// ----------------------------------------------------------
// msg002 Message 02
// ----------------------------------------------------------
      SET   ;
      R     DB2697.DBX  140.7;
      =     DB2697.DBX  141.4;

      CLR   ;
      =     DB2697.DBX  142.7;

// ----------------------------------------------------------
// msg003 Message 03
// ----------------------------------------------------------
      SET   ;
      R     DB2697.DBX  200.7;
      =     DB2697.DBX  201.4;

      CLR   ;
      =     DB2697.DBX  202.7;

NETWORK
TITLE =Sequence organisation

      CLR   ;
      =     M    122.2;

// SFM supply ----------------------------------------------------------------

// analog value to SFM Heißwasser-Wärmetauscher1 TT01 -----------------------
      L     DB2693.DBD  146;
      T     DB1691.DBD 1122; // !!! insert correct SFM !!!

// sequencer ----------------------------------------------------------------
      A     DB1693.DBX   43.1;
      S     DB1693.DBX   97.3;

      CALL FC    40 (
           UnitNo                   := #UnitNo);

NETWORK
TITLE =Auto / Manual

      SET   ;
      AN    M    122.2;
      JC    MODE;
      AN    M    120.1;

// assign actuator mode
      AN    M    120.1;
      =     DB2690.DBX 1545.4;
      =     DB2690.DBX 1625.4;
      =     DB2690.DBX 1705.4;
      =     DB2690.DBX 1785.4;
      =     DB2690.DBX 1865.4;
      =     DB2690.DBX 1945.4;
      =     DB2690.DBX 2025.4;
      =     DB2690.DBX 2105.4;
      =     DB2690.DBX 2185.4;
      =     DB2690.DBX 2265.4;
      =     DB2690.DBX 2345.4;
      =     DB2690.DBX 2425.4;
      =     DB2690.DBX 2505.4;
      =     DB2690.DBX 2585.4;
      =     DB2690.DBX 2665.4;
      =     DB2690.DBX 2745.4;
      =     DB2690.DBX 2825.4;
      =     DB2690.DBX 2905.4;
      =     DB2690.DBX 2985.4;
      =     DB2690.DBX 3065.4;
      =     DB2690.DBX 3145.4;
      =     DB2690.DBX 3225.4;



MODE: SET   ;

NETWORK
TITLE =A9_RR1 Reinigungsrücklauf Anlage 9 zu Kreis 1
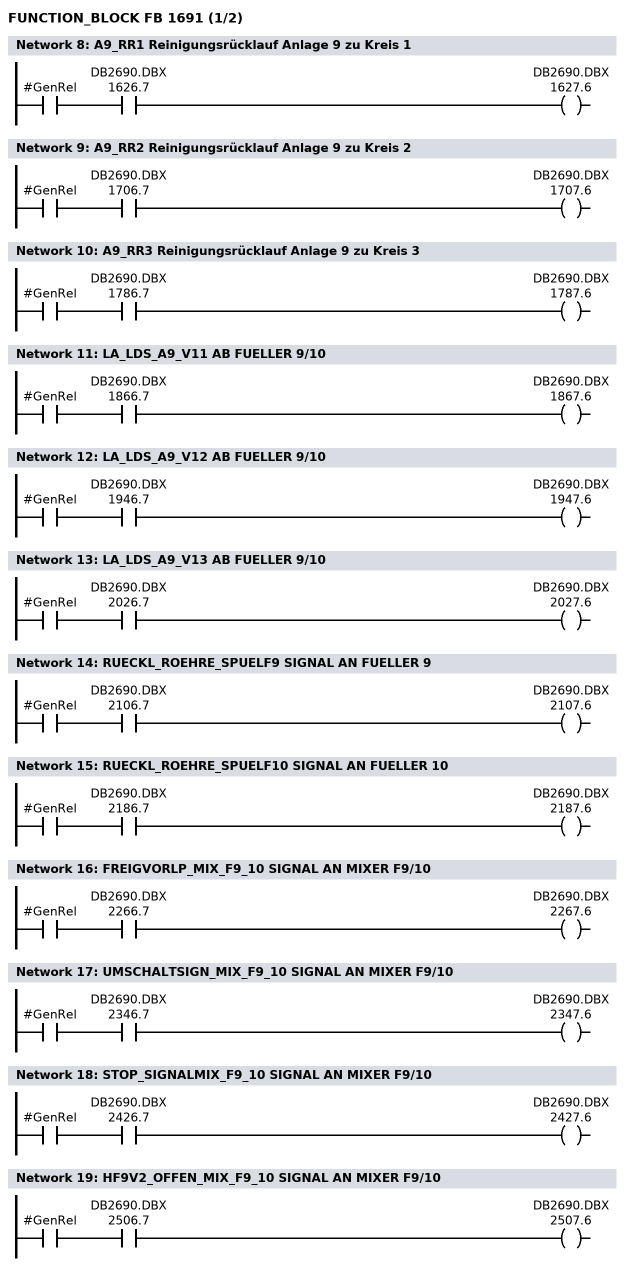

      A     #GenRel;
      A     DB2690.DBX 1626.7;
      =     DB2690.DBX 1627.6;
NETWORK
TITLE =A9_RR2 Reinigungsrücklauf Anlage 9 zu Kreis 2

      A     #GenRel;
      A     DB2690.DBX 1706.7;
      =     DB2690.DBX 1707.6;
NETWORK
TITLE =A9_RR3 Reinigungsrücklauf Anlage 9 zu Kreis 3

      A     #GenRel;
      A     DB2690.DBX 1786.7;
      =     DB2690.DBX 1787.6;
NETWORK
TITLE =LA_LDS_A9_V11 AB FUELLER 9/10

      A     #GenRel;
      A     DB2690.DBX 1866.7;
      =     DB2690.DBX 1867.6;
NETWORK
TITLE =LA_LDS_A9_V12 AB FUELLER 9/10

      A     #GenRel;
      A     DB2690.DBX 1946.7;
      =     DB2690.DBX 1947.6;
NETWORK
TITLE =LA_LDS_A9_V13 AB FUELLER 9/10

      A     #GenRel;
      A     DB2690.DBX 2026.7;
      =     DB2690.DBX 2027.6;
NETWORK
TITLE =RUECKL_ROEHRE_SPUELF9 SIGNAL AN FUELLER 9

      A     #GenRel;
      A     DB2690.DBX 2106.7;
      =     DB2690.DBX 2107.6;
NETWORK
TITLE =RUECKL_ROEHRE_SPUELF10 SIGNAL AN FUELLER 10

      A     #GenRel;
      A     DB2690.DBX 2186.7;
      =     DB2690.DBX 2187.6;
NETWORK
TITLE =FREIGVORLP_MIX_F9_10 SIGNAL AN MIXER F9/10

      A     #GenRel;
      A     DB2690.DBX 2266.7;
      =     DB2690.DBX 2267.6;
NETWORK
TITLE =UMSCHALTSIGN_MIX_F9_10 SIGNAL AN MIXER F9/10

      A     #GenRel;
      A     DB2690.DBX 2346.7;
      =     DB2690.DBX 2347.6;
NETWORK
TITLE =STOP_SIGNALMIX_F9_10 SIGNAL AN MIXER F9/10

      A     #GenRel;
      A     DB2690.DBX 2426.7;
      =     DB2690.DBX 2427.6;
NETWORK
TITLE =HF9V2_OFFEN_MIX_F9_10 SIGNAL AN MIXER F9/10

      A     #GenRel;
      A     DB2690.DBX 2506.7;
      =     DB2690.DBX 2507.6;
NETWORK
TITLE =FREIGVORLP_KASK_F9_10 SIGNAL AN MIXER F9/10
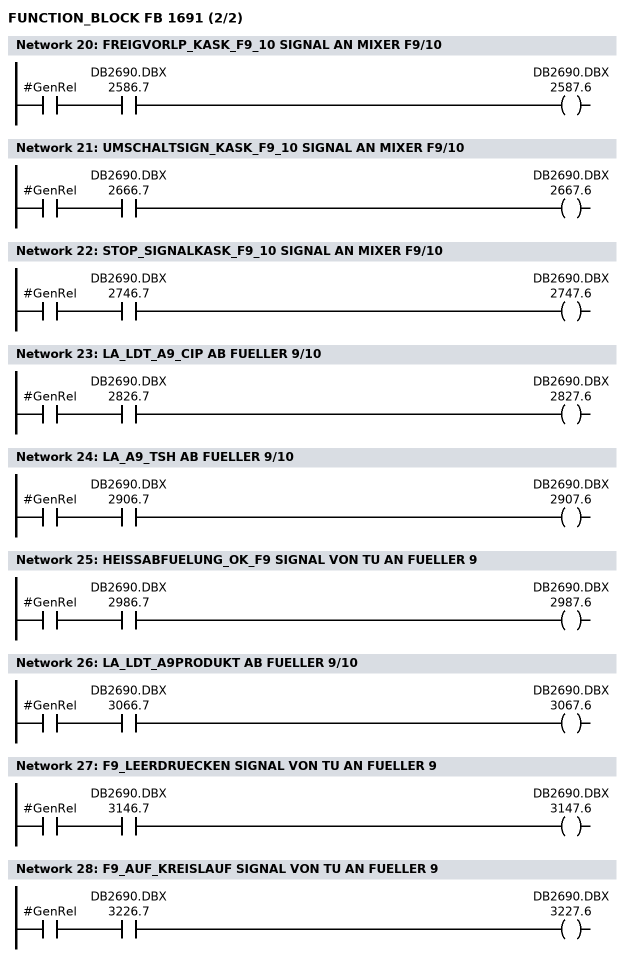

      A     #GenRel;
      A     DB2690.DBX 2586.7;
      =     DB2690.DBX 2587.6;
NETWORK
TITLE =UMSCHALTSIGN_KASK_F9_10 SIGNAL AN MIXER F9/10

      A     #GenRel;
      A     DB2690.DBX 2666.7;
      =     DB2690.DBX 2667.6;
NETWORK
TITLE =STOP_SIGNALKASK_F9_10 SIGNAL AN MIXER F9/10

      A     #GenRel;
      A     DB2690.DBX 2746.7;
      =     DB2690.DBX 2747.6;
NETWORK
TITLE =LA_LDT_A9_CIP AB FUELLER 9/10

      A     #GenRel;
      A     DB2690.DBX 2826.7;
      =     DB2690.DBX 2827.6;
NETWORK
TITLE =LA_A9_TSH AB FUELLER 9/10

      A     #GenRel;
      A     DB2690.DBX 2906.7;
      =     DB2690.DBX 2907.6;
NETWORK
TITLE =HEISSABFUELUNG_OK_F9 SIGNAL VON TU AN FUELLER 9

      A     #GenRel;
      A     DB2690.DBX 2986.7;
      =     DB2690.DBX 2987.6;
NETWORK
TITLE =LA_LDT_A9PRODUKT AB FUELLER 9/10

      A     #GenRel;
      A     DB2690.DBX 3066.7;
      =     DB2690.DBX 3067.6;
NETWORK
TITLE =F9_LEERDRUECKEN SIGNAL VON TU AN FUELLER 9

      A     #GenRel;
      A     DB2690.DBX 3146.7;
      =     DB2690.DBX 3147.6;
NETWORK
TITLE =F9_AUF_KREISLAUF SIGNAL VON TU AN FUELLER 9

      A     #GenRel;
      A     DB2690.DBX 3226.7;
      =     DB2690.DBX 3227.6;
END_FUNCTION_BLOCK

FUNCTION_BLOCK FB 1700
TITLE =U070: Abfüllanlage 10
FAMILY : BOTEC_F1
NAME : U070A
VERSION : 2.1


VAR_TEMP
  EStopOK : BOOL ;	//auxiliary flag
  CIP : BOOL ;	//CIP Program Selected
  xTmp : BOOL ;	//Temporary Bool(free for general use)
  DummyBool : BOOL ;	//Temporary Bool(free for general use)
  UnitNo : INT ;	//unit number
  UnitFB : INT ;	//unit expansion FB number
  rTmp : REAL ;	//Temporary REAL (free for general use)
  iTmp : INT ;	//Temporary INT (free for general use)
  DummyInt : INT ;	//Temporary INT (free for general use)
  dTmp : DINT ;	//Temporary DINT (free for general use)
END_VAR
BEGIN
NETWORK
TITLE =general

      CLR   ;
      =     #xTmp;
      =     #EStopOK;

      L     DB1700.DBW    0;
      T     #UnitNo;
      L     DB1700.DBW    2;
      T     #UnitFB;

NETWORK
TITLE =Universal value

      NOP   0;
// unv001 UnV 001 Process Status
      CALL FC    27 (
           UnitNo                   := #UnitNo,
           UnVRec                   := DB2705.unv001,
           ValExt                   := DB2705.DBD  234);

// unv002 UnV 002 Universal Value 02
      CALL FC    27 (
           UnitNo                   := #UnitNo,
           UnVRec                   := DB2705.unv002,
           ValExt                   := DB2705.DBD  362);

// unv003 UnV 003 Universal Value 03
      CALL FC    27 (
           UnitNo                   := #UnitNo,
           UnVRec                   := DB2705.unv003,
           ValExt                   := DB2705.DBD  490);

// unv004 UnV 004 Universal Value 04
      CALL FC    27 (
           UnitNo                   := #UnitNo,
           UnVRec                   := DB2705.unv004,
           ValExt                   := DB2705.DBD  618);

NETWORK
TITLE =special inputs

      NOP   0;
// LS_LLL_A10 SpI 001 LS_LLL_A10
      CALL FC    14 (
           UnitNo                   := #UnitNo,
           SpIRec                   := DB2701.LS_LLL_A10,
           SpIBit                   := I     62.3);

// TS_HL_ANL10 SpI 002 TS_HL_ANL10
      CALL FC    14 (
           UnitNo                   := #UnitNo,
           SpIRec                   := DB2701.TS_HL_ANL10,
           SpIBit                   := I     62.1);

// DT_A10_START SpI 003 DT_A10_START
      CALL FC    14 (
           UnitNo                   := #UnitNo,
           SpIRec                   := DB2701.DT_A10_START,
           SpIBit                   := I     53.4);

// DT_A10_STOP SpI 004 DT_A10_STOP
      CALL FC    14 (
           UnitNo                   := #UnitNo,
           SpIRec                   := DB2701.DT_A10_STOP,
           SpIBit                   := I     53.5);

// BETRIEB_F10 SpI 005 BETRIEB_F10
      CALL FC    14 (
           UnitNo                   := #UnitNo,
           SpIRec                   := DB2701.BETRIEB_F10,
           SpIBit                   := I     62.5);

// BETRIEB_MIX_LKASKADE_F10 SpI 006 BETRIEB_MIX_LKASKADE_F10
      CALL FC    14 (
           UnitNo                   := #UnitNo,
           SpIRec                   := DB2701.BETRIEB_MIX_LKASKADE_F10,
           SpIBit                   := I     62.7);

// KASK_ANFORDERUNG_PUMPE SpI 007 KASK_ANFORDERUNG_PUMPE
      CALL FC    14 (
           UnitNo                   := #UnitNo,
           SpIRec                   := DB2701.KASK_ANFORDERUNG_PUMPE,
           SpIBit                   := I    123.3);

// RM_RWPA10 SpI 008 RM_RWPA10
      CALL FC    14 (
           UnitNo                   := #UnitNo,
           SpIRec                   := DB2701.RM_RWPA10,
           SpIBit                   := I    123.4);

// KAS_WEGFREIGABE_10_L9 SpI 009 KAS_WEGFREIGABE_10_L9
      CALL FC    14 (
           UnitNo                   := #UnitNo,
           SpIRec                   := DB2701.KAS_WEGFREIGABE_10_L9,
           SpIBit                   := I    123.5);

// KAS_WEGFREIGABE_10_L10 SpI 010 KAS_WEGFREIGABE_10_L10
      CALL FC    14 (
           UnitNo                   := #UnitNo,
           SpIRec                   := DB2701.KAS_WEGFREIGABE_10_L10,
           SpIBit                   := I    123.6);

NETWORK
TITLE =messages

      NOP   0;
// msg001 Msg 001 Message 01
      CALL FC    16 (
           UnitNo                   := #UnitNo,
           MsgRec                   := DB2707.msg001,
           MsgBit                   := DB2707.DBX   82.7);

// msg002 Msg 002 Message 02
      CALL FC    16 (
           UnitNo                   := #UnitNo,
           MsgRec                   := DB2707.msg002,
           MsgBit                   := DB2707.DBX  142.7);

// msg003 Msg 003 Message 03
      CALL FC    16 (
           UnitNo                   := #UnitNo,
           MsgRec                   := DB2707.msg003,
           MsgBit                   := DB2707.DBX  202.7);

NETWORK
TITLE =unit supply

      UC    FB [#UnitFB];

NETWORK
TITLE =A10_RR1  Reinigungsrücklauf Anlage 10 zu Kreis 1
// Act 020
// Box           : VSRR1-3
// Input address : I84.6
// Output address: Q84.6
      CALL FC    70 (
           UnitNo                   := #UnitNo,
           ActRec                   := DB2700.A10_RR1,
           Typ                      := 1,
           FBa                      := #xTmp,
           FBa2                     := I     84.6,
           Out                      := Q     84.6);

NETWORK
TITLE =A10_RR2  Reinigungsrücklauf Anlage 10 zu Kreis 2
// Act 021
// Box           : VSRR1-3
// Input address : I84.7
// Output address: Q84.7
      CALL FC    70 (
           UnitNo                   := #UnitNo,
           ActRec                   := DB2700.A10_RR2,
           Typ                      := 1,
           FBa                      := #xTmp,
           FBa2                     := I     84.7,
           Out                      := Q     84.7);

NETWORK
TITLE =A10_RR3  Reinigungsrücklauf Anlage 10 zu Kreis 3
// Act 022
// Box           : VSRR1-3
// Input address : I85.0
// Output address: Q85.0
      CALL FC    70 (
           UnitNo                   := #UnitNo,
           ActRec                   := DB2700.A10_RR3,
           Typ                      := 1,
           FBa                      := #xTmp,
           FBa2                     := I     85.0,
           Out                      := Q     85.0);

NETWORK
TITLE =LA_LDS_A10V13  LA_LDS_A10V13
// Act 023
// Box           : S8 U8.2
// Input address : I53.1
// Output address: Q110.0
      CALL FC    70 (
           UnitNo                   := #UnitNo,
           ActRec                   := DB2700.LA_LDS_A10V13,
           Typ                      := 0,
           FBa                      := #xTmp,
           FBa2                     := I     53.1,
           Out                      := Q    110.0);

NETWORK
TITLE =LA_LDT_A10PRODUKT  LA_LDT_A10PRODUKT
// Act 024
// Box           : S8 U8.2
// Input address : I53.2
// Output address: Q110.1
      CALL FC    70 (
           UnitNo                   := #UnitNo,
           ActRec                   := DB2700.LA_LDT_A10PRODUKT,
           Typ                      := 0,
           FBa                      := #xTmp,
           FBa2                     := I     53.2,
           Out                      := Q    110.1);

NETWORK
TITLE =LA_LDT_A10CIP  LA_LDT_A10CIP
// Act 025
// Box           : S8 U8.2
// Input address : I53.3
// Output address: Q110.2
      CALL FC    70 (
           UnitNo                   := #UnitNo,
           ActRec                   := DB2700.LA_LDT_A10CIP,
           Typ                      := 0,
           FBa                      := #xTmp,
           FBa2                     := I     53.3,
           Out                      := Q    110.2);

NETWORK
TITLE =LA_A10TSH  LA_A10TSH
// Act 026
// Box           : S8 U8.2
// Output address: Q110.3
      CALL FC    70 (
           UnitNo                   := #UnitNo,
           ActRec                   := DB2700.LA_A10TSH,
           Typ                      := 0,
           FBa                      := #xTmp,
           FBa2                     := #xTmp,
           Out                      := Q    110.3);

NETWORK
TITLE =LA_STOERUNG_CIP  LA_STOERUNG_CIP
// Act 027
// Box           : S8 U8.2
// Output address: Q110.4
      CALL FC    70 (
           UnitNo                   := #UnitNo,
           ActRec                   := DB2700.LA_STOERUNG_CIP,
           Typ                      := 0,
           FBa                      := #xTmp,
           FBa2                     := #xTmp,
           Out                      := Q    110.4);

NETWORK
TITLE =LA_ALARML9_10  LA_ALARML9_10
// Act 028
// Box           : S8 U8.2
// Output address: Q110.5
      CALL FC    70 (
           UnitNo                   := #UnitNo,
           ActRec                   := DB2700.LA_ALARML9_10,
           Typ                      := 0,
           FBa                      := #xTmp,
           FBa2                     := #xTmp,
           Out                      := Q    110.5);

NETWORK
TITLE =LA_LDS_A10V11  LA_LDS_A10V11
// Act 029
// Box           : S8 U8.2
// Input address : I52.7
// Output address: Q110.6
      CALL FC    70 (
           UnitNo                   := #UnitNo,
           ActRec                   := DB2700.LA_LDS_A10V11,
           Typ                      := 0,
           FBa                      := #xTmp,
           FBa2                     := I     52.7,
           Out                      := Q    110.6);

NETWORK
TITLE =LA_LDS_A10V12  LA_LDS_A10V12
// Act 030
// Box           : S8 U8.2
// Input address : I53.0
// Output address: Q110.7
      CALL FC    70 (
           UnitNo                   := #UnitNo,
           ActRec                   := DB2700.LA_LDS_A10V12,
           Typ                      := 0,
           FBa                      := #xTmp,
           FBa2                     := I     53.0,
           Out                      := Q    110.7);

NETWORK
TITLE =UMSCHALTSIGN_KASK_F9_10  UMSCHALTSIGN_KASK_F9_10
// Act 031
// Box           : S8 U8.2
// Output address: Q41.6
      CALL FC    70 (
           UnitNo                   := #UnitNo,
           ActRec                   := DB2700.UMSCHALTSIGN_KASK_F9_10,
           Typ                      := 0,
           FBa                      := #xTmp,
           FBa2                     := #xTmp,
           Out                      := Q     41.6);

NETWORK
TITLE =STOP_SIGNALKASK_F9_10  STOP_SIGNALKASK_F9_10
// Act 032
// Box           : S8 U8.2
// Output address: Q41.7
      CALL FC    70 (
           UnitNo                   := #UnitNo,
           ActRec                   := DB2700.STOP_SIGNALKASK_F9_10,
           Typ                      := 0,
           FBa                      := #xTmp,
           FBa2                     := #xTmp,
           Out                      := Q     41.7);

END_FUNCTION_BLOCK

FUNCTION_BLOCK FB 1701
TITLE =U070: Packaging Plant 10
FAMILY : BOTEC_F1
NAME : UniE
VERSION : 1.2


VAR_TEMP
  CIP : BOOL ;	//CIP active
  UNIM : BOOL ;	//Unit Not In Maintenance
  GenRel : BOOL ;	//general OK (emergency and maintenance OK)
  EStopOK : BOOL ;	//emergency OK
  UnitNo : INT ;	//unit number
  xTmp : BOOL ;	//Temporary Bool
  iTmp : INT ;	//Temporary INT
  rTmp : REAL ;	//Temporary REAL
  dTmp : DINT ;	//Temporary DINT (free for general use)
  RetValInt : INT ;	//return value
END_VAR
BEGIN
NETWORK
TITLE =General

      SET   ;
// Simulation ---------------------------------------------------------------
      A     DB1701.DBX 1357.7;
      CC    FB  1709; // "U070Sim"
      A     DB1701.DBX   17.3;
      =     DB1701.DBX 1357.7; //Help bit for simulation

// get unit number ----------------------------------------------------------
      L     DB1700.DBW    0;
      T     #UnitNo;

// CIP ----------------------------------------------------------------------
      L     DB1701.DBD   54;
      L     0;
      <D    ;
      =     #CIP;

// emergency OK -------------------------------------------------------------
      A     DB1705.DBX   27.0; //Emergency Stop OK
      =     #EStopOK;

// Write Unit in Maintenance ------------------------------------------------

      AN    DB1701.DBX   69.7;
      =     #UNIM;

// emergency and maintenance OK ---------------------------------------------
      A     #EStopOK;
      A     #UNIM;
      =     #GenRel;

// communication ------------------------------------------------------------
      UC    FB  1705; // U070Com

NETWORK
TITLE =Universal Value

      NOP   0;

// ----------------------------------------------------------
// unv001 Process Status
// ----------------------------------------------------------
// process value to UnV
//      L     0.000000e+000
//      T     "U070UnVD".unv001.ValExt

// ----------------------------------------------------------
// unv002 Universal Value 02
// ----------------------------------------------------------
// process value to UnV
//      L     0.000000e+000
//      T     "U070UnVD".unv002.ValExt

// ----------------------------------------------------------
// unv003 Universal Value 03
// ----------------------------------------------------------
// process value to UnV
//      L     0.000000e+000
//      T     "U070UnVD".unv003.ValExt

// ----------------------------------------------------------
// unv004 Universal Value 04
// ----------------------------------------------------------
// process value to UnV
//      L     0.000000e+000
//      T     "U070UnVD".unv004.ValExt

NETWORK
TITLE =Special Input

      NOP   0;

// ----------------------------------------------------------
// LS_LLL_A10 SIGNAL VON FUELLER 10
// ----------------------------------------------------------
//      A     "U070SeqD".Seq.Step0
//      =     "U070SpID".LS_LLL_A10.EAl
//      SET
//      =     "U070SpID".LS_LLL_A10.Pre

// ----------------------------------------------------------
// TS_HL_ANL10
// ----------------------------------------------------------
//      A     "U070SeqD".Seq.Step0
//      =     "U070SpID".TS_HL_ANL10.EAl
//      SET
//      =     "U070SpID".TS_HL_ANL10.Pre

// ----------------------------------------------------------
// DT_A10_START AB FUELLER 9/10
// ----------------------------------------------------------
//      CLR
//      =     "U070SpID".DT_A10_START.EAl
//      =     "U070SpID".DT_A10_START.Pre

// ----------------------------------------------------------
// DT_A10_STOP AB FUELLER 9/10
// ----------------------------------------------------------
//      CLR
//      =     "U070SpID".DT_A10_STOP.EAl
//      =     "U070SpID".DT_A10_STOP.Pre

// ----------------------------------------------------------
// BETRIEB_F10 SIGNAL VON FUELLER 10
// ----------------------------------------------------------
//      CLR
//      =     "U070SpID".BETRIEB_F10.EAl
//      =     "U070SpID".BETRIEB_F10.Pre

// ----------------------------------------------------------
// BETRIEB_MIX_LKASKADE_F10 SIGNAL VON FUELLER 10
// ----------------------------------------------------------
//      CLR
//      =     "U070SpID".BETRIEB_MIX_LKASKADE_F10.EAl
//      =     "U070SpID".BETRIEB_MIX_LKASKADE_F10.Pre

// ----------------------------------------------------------
// KASK_ANFORDERUNG_PUMPE SIGNAL VON KASKADE
// ----------------------------------------------------------
//      CLR
//      =     "U070SpID".KASK_ANFORDERUNG_PUMPE.EAl
//      =     "U070SpID".KASK_ANFORDERUNG_PUMPE.Pre

// ----------------------------------------------------------
// RM_RWPA10 SIGNAL VON MIXER F9/10
// ----------------------------------------------------------
      A     DB1701.DBX 1230.3;
      A     DB1701.DBX 1262.3;
      =     DB2701.DBX  501.4;
      =     DB2701.DBX  501.5;

// ----------------------------------------------------------
// KAS_WEGFREIGABE_10_L9 SIGNAL VON KASKADE F9/10
// ----------------------------------------------------------
//      CLR
//      =     "U070SpID".KAS_WEGFREIGABE_10_L9.EAl
//      =     "U070SpID".KAS_WEGFREIGABE_10_L9.Pre

// ----------------------------------------------------------
// KAS_WEGFREIGABE_10_L10 SIGNAL VON KASKADE F9/10
// ----------------------------------------------------------
//      CLR
//      =     "U070SpID".KAS_WEGFREIGABE_10_L10.EAl
//      =     "U070SpID".KAS_WEGFREIGABE_10_L10.Pre

NETWORK
TITLE =Messages

      NOP   0;

// ----------------------------------------------------------
// msg001 Message 01
// ----------------------------------------------------------
      SET   ;
      R     DB2707.DBX   80.7;
      =     DB2707.DBX   81.4;

      CLR   ;
      =     DB2707.DBX   82.7;

// ----------------------------------------------------------
// msg002 Message 02
// ----------------------------------------------------------
      SET   ;
      R     DB2707.DBX  140.7;
      =     DB2707.DBX  141.4;

      CLR   ;
      =     DB2707.DBX  142.7;

// ----------------------------------------------------------
// msg003 Message 03
// ----------------------------------------------------------
      SET   ;
      R     DB2707.DBX  200.7;
      =     DB2707.DBX  201.4;

      CLR   ;
      =     DB2707.DBX  202.7;

NETWORK
TITLE =Sequence organisation

      CLR   ;
      =     M    122.2;

// SFM supply ----------------------------------------------------------------

// sequencer ----------------------------------------------------------------
      A     DB1703.DBX   43.1;
      S     DB1703.DBX   97.3;

      CALL FC    40 (
           UnitNo                   := #UnitNo);

NETWORK
TITLE =Auto / Manual

      SET   ;
      AN    M    122.2;
      JC    MODE;
      AN    M    120.1;

// assign actuator mode
      AN    M    120.1;
      =     DB2700.DBX 1625.4;
      =     DB2700.DBX 1705.4;
      =     DB2700.DBX 1785.4;
      =     DB2700.DBX 1865.4;
      =     DB2700.DBX 1945.4;
      =     DB2700.DBX 2025.4;
      =     DB2700.DBX 2105.4;
      =     DB2700.DBX 2185.4;
      =     DB2700.DBX 2265.4;
      =     DB2700.DBX 2345.4;
      =     DB2700.DBX 2425.4;
      =     DB2700.DBX 2505.4;
      =     DB2700.DBX 2585.4;

MODE: SET   ;

NETWORK
TITLE =A10_RR1 Reinigungsrücklauf Anlage 10 zu Kreis 1
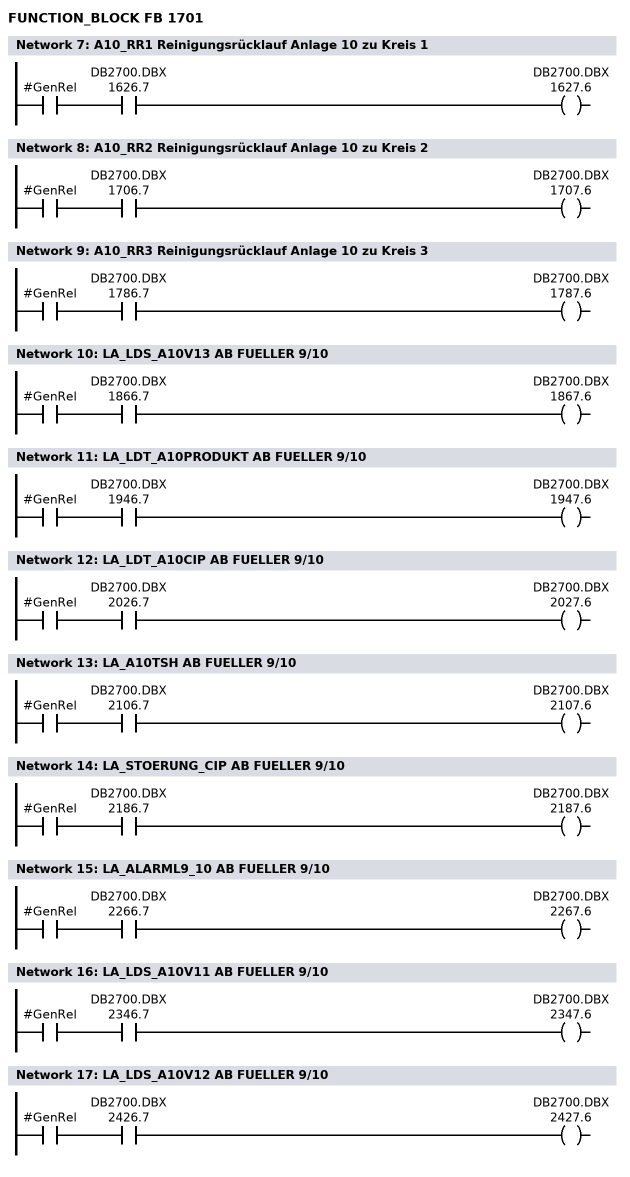

      A     #GenRel;
      A     DB2700.DBX 1626.7;
      =     DB2700.DBX 1627.6;
NETWORK
TITLE =A10_RR2 Reinigungsrücklauf Anlage 10 zu Kreis 2

      A     #GenRel;
      A     DB2700.DBX 1706.7;
      =     DB2700.DBX 1707.6;
NETWORK
TITLE =A10_RR3 Reinigungsrücklauf Anlage 10 zu Kreis 3

      A     #GenRel;
      A     DB2700.DBX 1786.7;
      =     DB2700.DBX 1787.6;
NETWORK
TITLE =LA_LDS_A10V13 AB FUELLER 9/10

      A     #GenRel;
      A     DB2700.DBX 1866.7;
      =     DB2700.DBX 1867.6;
NETWORK
TITLE =LA_LDT_A10PRODUKT AB FUELLER 9/10

      A     #GenRel;
      A     DB2700.DBX 1946.7;
      =     DB2700.DBX 1947.6;
NETWORK
TITLE =LA_LDT_A10CIP AB FUELLER 9/10

      A     #GenRel;
      A     DB2700.DBX 2026.7;
      =     DB2700.DBX 2027.6;
NETWORK
TITLE =LA_A10TSH AB FUELLER 9/10

      A     #GenRel;
      A     DB2700.DBX 2106.7;
      =     DB2700.DBX 2107.6;
NETWORK
TITLE =LA_STOERUNG_CIP AB FUELLER 9/10

      A     #GenRel;
      A     DB2700.DBX 2186.7;
      =     DB2700.DBX 2187.6;
NETWORK
TITLE =LA_ALARML9_10 AB FUELLER 9/10

      A     #GenRel;
      A     DB2700.DBX 2266.7;
      =     DB2700.DBX 2267.6;
NETWORK
TITLE =LA_LDS_A10V11 AB FUELLER 9/10

      A     #GenRel;
      A     DB2700.DBX 2346.7;
      =     DB2700.DBX 2347.6;
NETWORK
TITLE =LA_LDS_A10V12 AB FUELLER 9/10

      A     #GenRel;
      A     DB2700.DBX 2426.7;
      =     DB2700.DBX 2427.6;
END_FUNCTION_BLOCK

FUNCTION_BLOCK FB 1710
TITLE =U071: Abfüllanlage 11
FAMILY : BOTEC_F1
NAME : U071A
VERSION : 2.1


VAR_TEMP
  EStopOK : BOOL ;	//auxiliary flag
  CIP : BOOL ;	//CIP Program Selected
  xTmp : BOOL ;	//Temporary Bool(free for general use)
  DummyBool : BOOL ;	//Temporary Bool(free for general use)
  UnitNo : INT ;	//unit number
  UnitFB : INT ;	//unit expansion FB number
  rTmp : REAL ;	//Temporary REAL (free for general use)
  iTmp : INT ;	//Temporary INT (free for general use)
  DummyInt : INT ;	//Temporary INT (free for general use)
  dTmp : DINT ;	//Temporary DINT (free for general use)
END_VAR
BEGIN
NETWORK
TITLE =general

      CLR   ;
      =     #xTmp;
      =     #EStopOK;

      L     DB1710.DBW    0;
      T     #UnitNo;
      L     DB1710.DBW    2;
      T     #UnitFB;

NETWORK
TITLE =Universal value

      NOP   0;
// unv001 UnV 001 Process Status
      CALL FC    27 (
           UnitNo                   := #UnitNo,
           UnVRec                   := DB2715.unv001,
           ValExt                   := DB2715.DBD  234);

// unv002 UnV 002 Universal Value 02
      CALL FC    27 (
           UnitNo                   := #UnitNo,
           UnVRec                   := DB2715.unv002,
           ValExt                   := DB2715.DBD  362);

// unv003 UnV 003 Universal Value 03
      CALL FC    27 (
           UnitNo                   := #UnitNo,
           UnVRec                   := DB2715.unv003,
           ValExt                   := DB2715.DBD  490);

// unv004 UnV 004 Universal Value 04
      CALL FC    27 (
           UnitNo                   := #UnitNo,
           UnVRec                   := DB2715.unv004,
           ValExt                   := DB2715.DBD  618);

NETWORK
TITLE =special inputs

      NOP   0;
// A9_FS1 SpI 001 geändert 07.11.01 A11 FS1 Stömungswächter
      CALL FC    14 (
           UnitNo                   := #UnitNo,
           SpIRec                   := DB2711.A9_FS1,
           SpIBit                   := I    177.0);

// A11_Fueller_laeuft SpI 002 Füller 11 läuft (Dauersignal)
      CALL FC    14 (
           UnitNo                   := #UnitNo,
           SpIRec                   := DB2711.A11_Fueller_laeuft,
           SpIBit                   := I    168.1);

// A11_Mixer_CIP_Bereit SpI 003 Mixer A 11 CIP-Bereitschaft (Dauersign)
      CALL FC    14 (
           UnitNo                   := #UnitNo,
           SpIRec                   := DB2711.A11_Mixer_CIP_Bereit,
           SpIBit                   := I    170.0);

// A11_Mixer_voll SpI 004 Mixer A 11 voll
      CALL FC    14 (
           UnitNo                   := #UnitNo,
           SpIRec                   := DB2711.A11_Mixer_voll,
           SpIBit                   := I    170.2);

// A11_Mixer_leer SpI 005 Mixer A 11 leer
      CALL FC    14 (
           UnitNo                   := #UnitNo,
           SpIRec                   := DB2711.A11_Mixer_leer,
           SpIBit                   := I    170.1);

// A11_Mixer_Anf_Sirup SpI 006 Mixer A 11 Anforderung Sirup
      CALL FC    14 (
           UnitNo                   := #UnitNo,
           SpIRec                   := DB2711.A11_Mixer_Anf_Sirup,
           SpIBit                   := I    170.3);

// A11_Fueller_CIP_Bereit SpI 007 Füller 11 CIP-Bereitschaft (Dauer)
      CALL FC    14 (
           UnitNo                   := #UnitNo,
           SpIRec                   := DB2711.A11_Fueller_CIP_Bereit,
           SpIBit                   := I    168.0);

// A11_Fueller_leer SpI 011 Füller 11 leer (Impuls)
      CALL FC    14 (
           UnitNo                   := #UnitNo,
           SpIRec                   := DB2711.A11_Fueller_leer,
           SpIBit                   := I    168.2);

// All_Fueller_voll SpI 012 Füller 11 voll (Impuls)
      CALL FC    14 (
           UnitNo                   := #UnitNo,
           SpIRec                   := DB2711.All_Fueller_voll,
           SpIBit                   := I    168.3);

NETWORK
TITLE =messages

      NOP   0;
// msg001 Msg 001 Message 01
      CALL FC    16 (
           UnitNo                   := #UnitNo,
           MsgRec                   := DB2717.msg001,
           MsgBit                   := DB2717.DBX   82.7);

// msg002 Msg 002 Message 02
      CALL FC    16 (
           UnitNo                   := #UnitNo,
           MsgRec                   := DB2717.msg002,
           MsgBit                   := DB2717.DBX  142.7);

// msg003 Msg 003 Message 03
      CALL FC    16 (
           UnitNo                   := #UnitNo,
           MsgRec                   := DB2717.msg003,
           MsgBit                   := DB2717.DBX  202.7);

NETWORK
TITLE =unit supply

      UC    FB [#UnitFB];

NETWORK
TITLE =A11_RP1  A11RP1 Anlage 11 Reinigungsrücklaufpumpe
// Act 001
// Box           : S6 U6.3
// Input address : I6.3
// Output address: Q6.3
      CALL FC    70 (
           UnitNo                   := #UnitNo,
           ActRec                   := DB2710.A11_RP1,
           Typ                      := 1,
           FBa                      := #xTmp,
           FBa2                     := I      6.3,
           Out                      := Q      6.3);

NETWORK
TITLE =F11_Maschine_Start  Füller 11 Maschine_Start
// Act 002
// Box           : FM-A11
// Output address: Q168.0
      CALL FC    70 (
           UnitNo                   := #UnitNo,
           ActRec                   := DB2710.F11_Maschine_Start,
           Typ                      := 0,
           FBa                      := #xTmp,
           FBa2                     := #xTmp,
           Out                      := Q    168.0);

NETWORK
TITLE =F11_Maschine_Stop  Füller 11 Maschine_Stop
// Act 003
// Box           : FM-A11
// Output address: Q168.1
      CALL FC    70 (
           UnitNo                   := #UnitNo,
           ActRec                   := DB2710.F11_Maschine_Stop,
           Typ                      := 0,
           FBa                      := #xTmp,
           FBa2                     := #xTmp,
           Out                      := #xTmp);

NETWORK
TITLE =F11_CIP_Kreislauf_o_puls  Füller 11 CIP-Kreisl. ohne puls
// Act 010
// Box           : FM-A11
// Output address: Q168.2
      CALL FC    70 (
           UnitNo                   := #UnitNo,
           ActRec                   := DB2710.F11_CIP_Kreislauf_o_puls,
           Typ                      := 0,
           FBa                      := #xTmp,
           FBa2                     := #xTmp,
           Out                      := Q    168.2);

NETWORK
TITLE =F11_CIP_Kreislauf_m_puls  Füller 11 CIP-Kreisl. mit puls
// Act 011
// Box           : FM-A11
// Output address: Q168.3
      CALL FC    70 (
           UnitNo                   := #UnitNo,
           ActRec                   := DB2710.F11_CIP_Kreislauf_m_puls,
           Typ                      := 0,
           FBa                      := #xTmp,
           FBa2                     := #xTmp,
           Out                      := Q    168.3);

NETWORK
TITLE =F11_Randvollstellung  Füller 11 Randvollstellung Desinfektion
// Act 012
// Box           : FM-A11
// Output address: Q168.4
      CALL FC    70 (
           UnitNo                   := #UnitNo,
           ActRec                   := DB2710.F11_Randvollstellung,
           Typ                      := 0,
           FBa                      := #xTmp,
           FBa2                     := #xTmp,
           Out                      := Q    168.4);

NETWORK
TITLE =F11_Klarspuel_o_CIP_Beh  Füller 11 Klarspülen ohne CIP-Behälter
// Act 013
// Box           : FM-A11
// Output address: Q168.5
      CALL FC    70 (
           UnitNo                   := #UnitNo,
           ActRec                   := DB2710.F11_Klarspuel_o_CIP_Beh,
           Typ                      := 0,
           FBa                      := #xTmp,
           FBa2                     := #xTmp,
           Out                      := Q    168.5);

NETWORK
TITLE =F11_Ausschub_m_Steriluft  Füller 11 Ausschub mit Sterrielluft
// Act 014
// Box           : FM-A11
// Output address: Q168.6
      CALL FC    70 (
           UnitNo                   := #UnitNo,
           ActRec                   := DB2710.F11_Ausschub_m_Steriluft,
           Typ                      := 0,
           FBa                      := #xTmp,
           FBa2                     := #xTmp,
           Out                      := Q    168.6);

NETWORK
TITLE =F11_Ausschub_m_CO2  Füller 11 Ausschub mit CO2
// Act 015
// Box           : FM-A11
// Output address: Q168.7
      CALL FC    70 (
           UnitNo                   := #UnitNo,
           ActRec                   := DB2710.F11_Ausschub_m_CO2,
           Typ                      := 0,
           FBa                      := #xTmp,
           FBa2                     := #xTmp,
           Out                      := Q    168.7);

NETWORK
TITLE =F11_Grundstellung_IMP  F11_Grungstellung_IMPULS
// Act 016
// Box           : FM-A11
// Output address: Q169.0
      CALL FC    70 (
           UnitNo                   := #UnitNo,
           ActRec                   := DB2710.F11_Grundstellung_IMP,
           Typ                      := 0,
           FBa                      := #xTmp,
           FBa2                     := #xTmp,
           Out                      := Q    169.0);

NETWORK
TITLE =F11_Drainagestellung_IMP  F11_Drainagestellung_IMPULS
// Act 017
// Box           : FM-A11
// Output address: Q169.1
      CALL FC    70 (
           UnitNo                   := #UnitNo,
           ActRec                   := DB2710.F11_Drainagestellung_IMP,
           Typ                      := 0,
           FBa                      := #xTmp,
           FBa2                     := #xTmp,
           Out                      := Q    169.1);

NETWORK
TITLE =F11_Bypass_IMP  F11_BYPASS_IMPULS
// Act 018
// Box           : FM-A11
// Output address: Q169.2
      CALL FC    70 (
           UnitNo                   := #UnitNo,
           ActRec                   := DB2710.F11_Bypass_IMP,
           Typ                      := 0,
           FBa                      := #xTmp,
           FBa2                     := #xTmp,
           Out                      := Q    169.2);

NETWORK
TITLE =A11_RR1  A11RR1 Ventil CIP Rücklauf Kreis 1 Anlage 11
// Act 020
// Box           : VSRR6-11
// Input address : I28.3
// Output address: Q28.3
      CALL FC    70 (
           UnitNo                   := #UnitNo,
           ActRec                   := DB2710.A11_RR1,
           Typ                      := 1,
           FBa                      := #xTmp,
           FBa2                     := I     28.3,
           Out                      := Q     28.3);

NETWORK
TITLE =A11_RR2  A11RR2 Ventil CIP Rücklauf Kreis 2 Anlage 11
// Act 021
// Box           : VSRR6-11
// Input address : I28.4
// Output address: Q28.4
      CALL FC    70 (
           UnitNo                   := #UnitNo,
           ActRec                   := DB2710.A11_RR2,
           Typ                      := 1,
           FBa                      := #xTmp,
           FBa2                     := I     28.4,
           Out                      := Q     28.4);

NETWORK
TITLE =A11_RR3  A11RR3 Ventil CIP Rücklauf Kreis 3 Anlage 11
// Act 022
// Box           : VSRR6-11
// Input address : I28.5
// Output address: Q28.5
      CALL FC    70 (
           UnitNo                   := #UnitNo,
           ActRec                   := DB2710.A11_RR3,
           Typ                      := 1,
           FBa                      := #xTmp,
           FBa2                     := I     28.5,
           Out                      := Q     28.5);

NETWORK
TITLE =M11_Grundstellung_IMP  Mixer A11 Sign. als Impuls
// Act 023
// Box           : FM-A11
// Output address: Q170.0
      CALL FC    70 (
           UnitNo                   := #UnitNo,
           ActRec                   := DB2710.M11_Grundstellung_IMP,
           Typ                      := 0,
           FBa                      := #xTmp,
           FBa2                     := #xTmp,
           Out                      := Q    170.0);

NETWORK
TITLE =M11_Drainagestellung_IMP  Mixer A11 Sign. als Impuls
// Act 024
// Box           : FM-A11
// Output address: Q170.1
      CALL FC    70 (
           UnitNo                   := #UnitNo,
           ActRec                   := DB2710.M11_Drainagestellung_IMP,
           Typ                      := 0,
           FBa                      := #xTmp,
           FBa2                     := #xTmp,
           Out                      := Q    170.1);

NETWORK
TITLE =M11_Ausspritzen_o_Ablauf  Mixer A11 Sign. als Impuls
// Act 025
// Box           : FM-A11
// Output address: Q170.2
      CALL FC    70 (
           UnitNo                   := #UnitNo,
           ActRec                   := DB2710.M11_Ausspritzen_o_Ablauf,
           Typ                      := 0,
           FBa                      := #xTmp,
           FBa2                     := #xTmp,
           Out                      := Q    170.2);

NETWORK
TITLE =M11_Ausspritzen_m_Ablauf  Mixer A11 Sign. als Impuls
// Act 026
// Box           : FM-A11
// Output address: Q170.3
      CALL FC    70 (
           UnitNo                   := #UnitNo,
           ActRec                   := DB2710.M11_Ausspritzen_m_Ablauf,
           Typ                      := 0,
           FBa                      := #xTmp,
           FBa2                     := #xTmp,
           Out                      := Q    170.3);

NETWORK
TITLE =M11_Fluten_o_Ablauf  Mixer A11 Sign. als Impuls
// Act 027
// Box           : FM-A11
// Output address: Q170.4
      CALL FC    70 (
           UnitNo                   := #UnitNo,
           ActRec                   := DB2710.M11_Fluten_o_Ablauf,
           Typ                      := 0,
           FBa                      := #xTmp,
           FBa2                     := #xTmp,
           Out                      := Q    170.4);

NETWORK
TITLE =M11_Fluten_m_Ablauf  Mixer A11 Sign. als Impuls
// Act 028
// Box           : FM-A11
// Output address: Q170.5
      CALL FC    70 (
           UnitNo                   := #UnitNo,
           ActRec                   := DB2710.M11_Fluten_m_Ablauf,
           Typ                      := 0,
           FBa                      := #xTmp,
           FBa2                     := #xTmp,
           Out                      := Q    170.5);

NETWORK
TITLE =M11_Randvollstellung  Mixer A11 Sign. als Impuls
// Act 029
// Box           : FM-A11
// Output address: Q170.6
      CALL FC    70 (
           UnitNo                   := #UnitNo,
           ActRec                   := DB2710.M11_Randvollstellung,
           Typ                      := 0,
           FBa                      := #xTmp,
           FBa2                     := #xTmp,
           Out                      := Q    170.6);

NETWORK
TITLE =M11_Abpumpen  Mixer A11 Sign. als Impuls
// Act 030
// Box           : FM-A11
// Output address: Q170.7
      CALL FC    70 (
           UnitNo                   := #UnitNo,
           ActRec                   := DB2710.M11_Abpumpen,
           Typ                      := 0,
           FBa                      := #xTmp,
           FBa2                     := #xTmp,
           Out                      := Q    170.7);

NETWORK
TITLE =M11_Klarspuelen  Mixer A11
// Act 031
// Box           : FM-A11
// Output address: Q171.0
      CALL FC    70 (
           UnitNo                   := #UnitNo,
           ActRec                   := DB2710.M11_Klarspuelen,
           Typ                      := 0,
           FBa                      := #xTmp,
           FBa2                     := #xTmp,
           Out                      := Q    171.0);

NETWORK
TITLE =VNI_MOLCH_verr_A11  SIGNAL AN VNI Molch verriegelt an Anlage11
// Act 043
// Box           : AB-SK
// Output address: Q183.5
      CALL FC    70 (
           UnitNo                   := #UnitNo,
           ActRec                   := DB2710.VNI_MOLCH_verr_A11,
           Typ                      := 0,
           FBa                      := #xTmp,
           FBa2                     := #xTmp,
           Out                      := Q    183.5);

NETWORK
TITLE =VNI_MOLCH_Sender_A11  VNI Molch an Sendestation (SK)
// Act 044
// Box           : AB-SK
// Output address: Q183.6
      CALL FC    70 (
           UnitNo                   := #UnitNo,
           ActRec                   := DB2710.VNI_MOLCH_Sender_A11,
           Typ                      := 0,
           FBa                      := #xTmp,
           FBa2                     := #xTmp,
           Out                      := Q    183.6);

NETWORK
TITLE =VNI_MOLCH_Empfang_A11  VNI Molch an Empfangsstation (M11)
// Act 045
// Box           : AB-SK
// Output address: Q183.7
      CALL FC    70 (
           UnitNo                   := #UnitNo,
           ActRec                   := DB2710.VNI_MOLCH_Empfang_A11,
           Typ                      := 0,
           FBa                      := #xTmp,
           FBa2                     := #xTmp,
           Out                      := Q    183.7);

END_FUNCTION_BLOCK

FUNCTION_BLOCK FB 1711
TITLE =U071: Packaging Plant 11
FAMILY : BOTEC_F1
NAME : UniE
VERSION : 1.2


VAR_TEMP
  CIP : BOOL ;	//CIP active
  UNIM : BOOL ;	//Unit Not In Maintenance
  GenRel : BOOL ;	//general OK (emergency and maintenance OK)
  EStopOK : BOOL ;	//emergency OK
  UnitNo : INT ;	//unit number
  xTmp : BOOL ;	//Temporary Bool
  iTmp : INT ;	//Temporary INT
  rTmp : REAL ;	//Temporary REAL
  dTmp : DINT ;	//Temporary DINT (free for general use)
  RetValInt : INT ;	//return value
END_VAR
BEGIN
NETWORK
TITLE =General

      SET   ;
// Simulation ---------------------------------------------------------------
      A     DB1711.DBX 1357.7;
      CC    FB  1719; // "U071Sim"
      A     DB1711.DBX   17.3;
      =     DB1711.DBX 1357.7; //Help bit for simulation

// get unit number ----------------------------------------------------------
      L     DB1710.DBW    0;
      T     #UnitNo;

// CIP ----------------------------------------------------------------------
      L     DB1711.DBD   54;
      L     0;
      <D    ;
      =     #CIP;

// emergency OK -------------------------------------------------------------
      A     DB1715.DBX   27.0; //Emergency Stop OK
      =     #EStopOK;

// Write Unit in Maintenance ------------------------------------------------

      AN    DB1711.DBX   69.7;
      =     #UNIM;

// emergency and maintenance OK ---------------------------------------------
      A     #EStopOK;
      A     #UNIM;
      =     #GenRel;

// communication ------------------------------------------------------------
      UC    FB  1715; // U071Com

NETWORK
TITLE =Universal Value

      NOP   0;

// ----------------------------------------------------------
// unv001 Process Status
// ----------------------------------------------------------
// process value to UnV
//      L     0.000000e+000
//      T     "U071UnVD".unv001.ValExt

// ----------------------------------------------------------
// unv002 Universal Value 02
// ----------------------------------------------------------
// process value to UnV
//      L     0.000000e+000
//      T     "U071UnVD".unv002.ValExt

// ----------------------------------------------------------
// unv003 Universal Value 03
// ----------------------------------------------------------
// process value to UnV
//      L     0.000000e+000
//      T     "U071UnVD".unv003.ValExt

// ----------------------------------------------------------
// unv004 Universal Value 04
// ----------------------------------------------------------
// process value to UnV
//      L     0.000000e+000
//      T     "U071UnVD".unv004.ValExt

NETWORK
TITLE =Special Input

      NOP   0;

// ----------------------------------------------------------
// A11_Fueller_laeuft Füller 11 läuft (Dauersignal)
// ----------------------------------------------------------
//      CLR
//      =     "U071SpID".A11_Fueller_laeuft.EAl
//      =     "U071SpID".A11_Fueller_laeuft.Pre

// ----------------------------------------------------------
// A11_Mixer_CIP_Bereit Mixer A 11 CIP-Bereitschaft (Dauersign)
// ----------------------------------------------------------
//      CLR
//      =     "U071SpID".A11_Mixer_CIP_Bereit.EAl
//      =     "U071SpID".A11_Mixer_CIP_Bereit.Pre

// ----------------------------------------------------------
// A11_Mixer_voll Mixer A 11 voll
// ----------------------------------------------------------
//      CLR
//      =     "U071SpID".A11_Mixer_voll.EAl
//      =     "U071SpID".A11_Mixer_voll.Pre

// ----------------------------------------------------------
// A11_Mixer_leer Mixer A 11 leer
// ----------------------------------------------------------
//      CLR
//      =     "U071SpID".A11_Mixer_leer.EAl
//      =     "U071SpID".A11_Mixer_leer.Pre

// ----------------------------------------------------------
// A11_Mixer_Anf_Sirup Mixer A 11 Anforderung Sirup
// ----------------------------------------------------------
//      CLR
//      =     "U071SpID".A11_Mixer_Anf_Sirup.EAl
//      =     "U071SpID".A11_Mixer_Anf_Sirup.Pre

// ----------------------------------------------------------
// A11_Fueller_leer Füller 11 leer (Impuls)
// ----------------------------------------------------------
//      CLR
//      =     "U071SpID".A11_Fueller_leer.EAl
//      =     "U071SpID".A11_Fueller_leer.Pre

// ----------------------------------------------------------
// All_Fueller_voll Füller 11 voll (Impuls)
// ----------------------------------------------------------
//      CLR
//      =     "U071SpID".All_Fueller_voll.EAl
//      =     "U071SpID".All_Fueller_voll.Pre

NETWORK
TITLE =Messages

      NOP   0;

// ----------------------------------------------------------
// msg001 Message 01
// ----------------------------------------------------------
      SET   ;
      R     DB2717.DBX   80.7;
      =     DB2717.DBX   81.4;

      CLR   ;
      =     DB2717.DBX   82.7;

// ----------------------------------------------------------
// msg002 Message 02
// ----------------------------------------------------------
      SET   ;
      R     DB2717.DBX  140.7;
      =     DB2717.DBX  141.4;

      CLR   ;
      =     DB2717.DBX  142.7;

// ----------------------------------------------------------
// msg003 Message 03
// ----------------------------------------------------------
      SET   ;
      R     DB2717.DBX  200.7;
      =     DB2717.DBX  201.4;

      CLR   ;
      =     DB2717.DBX  202.7;

NETWORK
TITLE =Sequence organisation

      CLR   ;
      =     M    122.2;

// SFM supply ----------------------------------------------------------------

// sequencer ----------------------------------------------------------------
      A     DB1713.DBX   43.1;
      S     DB1713.DBX   97.3;

      CALL FC    40 (
           UnitNo                   := #UnitNo);

NETWORK
TITLE =Auto / Manual

      SET   ;
      AN    M    122.2;
      JC    MODE;
      AN    M    120.1;

// assign actuator mode
      AN    M    120.1;
      =     DB2710.DBX  105.4;
      =     DB2710.DBX  185.4;
      S     DB2710.DBX  265.4;
      =     DB2710.DBX  825.4;
      =     DB2710.DBX  905.4;
      =     DB2710.DBX  985.4;
      =     DB2710.DBX 1065.4;
      =     DB2710.DBX 1145.4;
      =     DB2710.DBX 1225.4;
      =     DB2710.DBX 1305.4;
      =     DB2710.DBX 1385.4;
      =     DB2710.DBX 1465.4;
      =     DB2710.DBX 1625.4;
      =     DB2710.DBX 1705.4;
      =     DB2710.DBX 1785.4;

      =     DB2710.DBX 1865.4;
      =     DB2710.DBX 1945.4;
      =     DB2710.DBX 2025.4;
      =     DB2710.DBX 2105.4;
      =     DB2710.DBX 2185.4;
      =     DB2710.DBX 2265.4;
      =     DB2710.DBX 2345.4;
      =     DB2710.DBX 2425.4;
      =     DB2710.DBX 2505.4;

      =     DB2710.DBX 3465.4;
      =     DB2710.DBX 3545.4;
      =     DB2710.DBX 3625.4;



MODE: SET   ;

NETWORK
TITLE =A11_RP1 A11RP1 Anlage 11 Reinigungsrücklaufpumpe
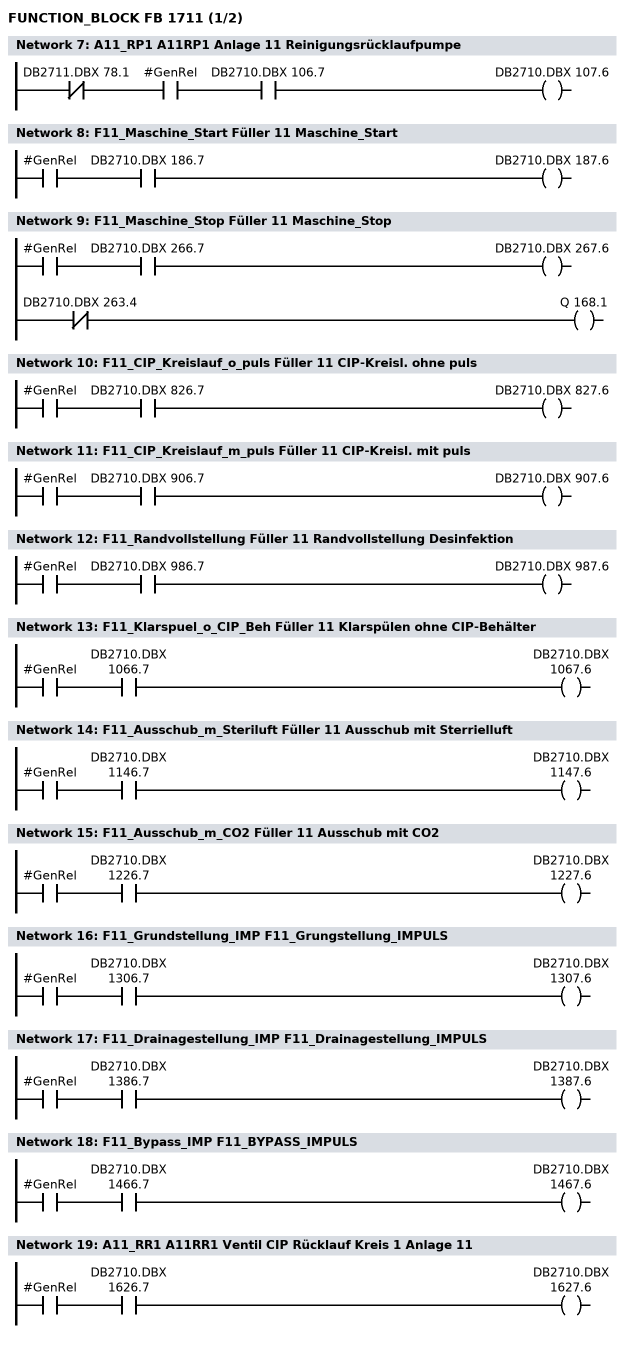

//      A     "U071SpID".A9_FS1.Sig
      AN    DB2711.DBX   78.1;

      A     #GenRel;
      A     DB2710.DBX  106.7;
      =     DB2710.DBX  107.6;
NETWORK
TITLE =F11_Maschine_Start Füller 11 Maschine_Start

      A     #GenRel;
      A     DB2710.DBX  186.7;
      =     DB2710.DBX  187.6;
NETWORK
TITLE =F11_Maschine_Stop Füller 11 Maschine_Stop

      A     #GenRel;
      A     DB2710.DBX  266.7;
      =     DB2710.DBX  267.6;

      AN    DB2710.DBX  263.4;
      =     Q    168.1;
NETWORK
TITLE =F11_CIP_Kreislauf_o_puls Füller 11 CIP-Kreisl. ohne puls

      A     #GenRel;
      A     DB2710.DBX  826.7;
      =     DB2710.DBX  827.6;
NETWORK
TITLE =F11_CIP_Kreislauf_m_puls Füller 11 CIP-Kreisl. mit puls

      A     #GenRel;
      A     DB2710.DBX  906.7;
      =     DB2710.DBX  907.6;
NETWORK
TITLE =F11_Randvollstellung Füller 11 Randvollstellung Desinfektion

      A     #GenRel;
      A     DB2710.DBX  986.7;
      =     DB2710.DBX  987.6;
NETWORK
TITLE =F11_Klarspuel_o_CIP_Beh Füller 11 Klarspülen ohne CIP-Behälter

      A     #GenRel;
      A     DB2710.DBX 1066.7;
      =     DB2710.DBX 1067.6;
NETWORK
TITLE =F11_Ausschub_m_Steriluft Füller 11 Ausschub mit Sterrielluft

      A     #GenRel;
      A     DB2710.DBX 1146.7;
      =     DB2710.DBX 1147.6;
NETWORK
TITLE =F11_Ausschub_m_CO2 Füller 11 Ausschub mit CO2

      A     #GenRel;
      A     DB2710.DBX 1226.7;
      =     DB2710.DBX 1227.6;
NETWORK
TITLE =F11_Grundstellung_IMP F11_Grungstellung_IMPULS

      A     #GenRel;
      A     DB2710.DBX 1306.7;
      =     DB2710.DBX 1307.6;
NETWORK
TITLE =F11_Drainagestellung_IMP F11_Drainagestellung_IMPULS

      A     #GenRel;
      A     DB2710.DBX 1386.7;
      =     DB2710.DBX 1387.6;
NETWORK
TITLE =F11_Bypass_IMP F11_BYPASS_IMPULS

      A     #GenRel;
      A     DB2710.DBX 1466.7;
      =     DB2710.DBX 1467.6;
NETWORK
TITLE =A11_RR1 A11RR1 Ventil CIP Rücklauf Kreis 1 Anlage 11

      A     #GenRel;
      A     DB2710.DBX 1626.7;
      =     DB2710.DBX 1627.6;
NETWORK
TITLE =A11_RR2 A11RR2 Ventil CIP Rücklauf Kreis 2 Anlage 11
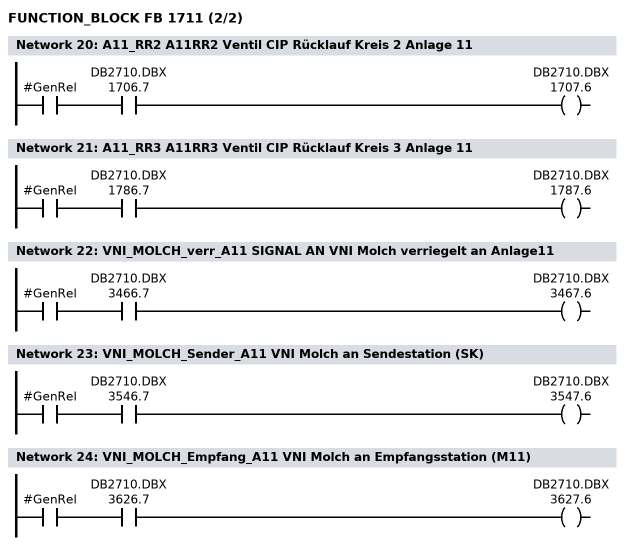

      A     #GenRel;
      A     DB2710.DBX 1706.7;
      =     DB2710.DBX 1707.6;
NETWORK
TITLE =A11_RR3 A11RR3 Ventil CIP Rücklauf Kreis 3 Anlage 11

      A     #GenRel;
      A     DB2710.DBX 1786.7;
      =     DB2710.DBX 1787.6;
NETWORK
TITLE =VNI_MOLCH_verr_A11 SIGNAL AN VNI Molch verriegelt an Anlage11

      A     #GenRel;
      A     DB2710.DBX 3466.7;
      =     DB2710.DBX 3467.6;
NETWORK
TITLE =VNI_MOLCH_Sender_A11 VNI Molch an Sendestation (SK)

      A     #GenRel;
      A     DB2710.DBX 3546.7;
      =     DB2710.DBX 3547.6;
NETWORK
TITLE =VNI_MOLCH_Empfang_A11 VNI Molch an Empfangsstation (M11)

      A     #GenRel;
      A     DB2710.DBX 3626.7;
      =     DB2710.DBX 3627.6;
END_FUNCTION_BLOCK

FUNCTION_BLOCK FB 1720
TITLE =U072: Abfüllanlage 12
FAMILY : BOTEC_F1
NAME : U072A
VERSION : 2.1


VAR_TEMP
  EStopOK : BOOL ;	//auxiliary flag
  CIP : BOOL ;	//CIP Program Selected
  xTmp : BOOL ;	//Temporary Bool(free for general use)
  DummyBool : BOOL ;	//Temporary Bool(free for general use)
  UnitNo : INT ;	//unit number
  UnitFB : INT ;	//unit expansion FB number
  rTmp : REAL ;	//Temporary REAL (free for general use)
  iTmp : INT ;	//Temporary INT (free for general use)
  DummyInt : INT ;	//Temporary INT (free for general use)
  dTmp : DINT ;	//Temporary DINT (free for general use)
END_VAR
BEGIN
NETWORK
TITLE =general

      CLR   ;
      =     #xTmp;
      =     #EStopOK;

      L     DB1720.DBW    0;
      T     #UnitNo;
      L     DB1720.DBW    2;
      T     #UnitFB;

NETWORK
TITLE =Universal value

      NOP   0;
// unv001 UnV 001 Process Status
      CALL FC    27 (
           UnitNo                   := #UnitNo,
           UnVRec                   := DB2725.unv001,
           ValExt                   := DB2725.DBD  234);

// unv002 UnV 002 Universal Value 02
      CALL FC    27 (
           UnitNo                   := #UnitNo,
           UnVRec                   := DB2725.unv002,
           ValExt                   := DB2725.DBD  362);

// unv003 UnV 003 Universal Value 03
      CALL FC    27 (
           UnitNo                   := #UnitNo,
           UnVRec                   := DB2725.unv003,
           ValExt                   := DB2725.DBD  490);

// unv004 UnV 004 Universal Value 04
      CALL FC    27 (
           UnitNo                   := #UnitNo,
           UnVRec                   := DB2725.unv004,
           ValExt                   := DB2725.DBD  618);

NETWORK
TITLE =special inputs

      NOP   0;
// A12_FS1 SpI 001 Anlage 12 Strömungswächter
      CALL FC    14 (
           UnitNo                   := #UnitNo,
           SpIRec                   := DB2721.A12_FS1,
           SpIBit                   := I    263.0);

// A12_FUELLER_LAEUFT SpI 002 Koppelsignal von Füller 12 Füller läuft (Dauersignal)
      CALL FC    14 (
           UnitNo                   := #UnitNo,
           SpIRec                   := DB2721.A12_FUELLER_LAEUFT,
           SpIBit                   := I    268.1);

// A12_MIXER_CIP_BEREIT SpI 003 Koppelsignal von Mixer 5 CIP-Bereitschaft (Dauersignal)
      CALL FC    14 (
           UnitNo                   := #UnitNo,
           SpIRec                   := DB2721.A12_MIXER_CIP_BEREIT,
           SpIBit                   := I    270.0);

// A12_MIXER_VOLL SpI 004 Koppelsignal von Mixer 5 Mixer voll
      CALL FC    14 (
           UnitNo                   := #UnitNo,
           SpIRec                   := DB2721.A12_MIXER_VOLL,
           SpIBit                   := I    270.1);

// A12_MIXER_LEER SpI 005 Koppelsignal von Mixer 5 Mixer leer
      CALL FC    14 (
           UnitNo                   := #UnitNo,
           SpIRec                   := DB2721.A12_MIXER_LEER,
           SpIBit                   := I    270.2);

// A12_MIXER_Anforderung SpI 006 Koppelsignal von Mixer 5 Anforderung Nachsp.
      CALL FC    14 (
           UnitNo                   := #UnitNo,
           SpIRec                   := DB2721.A12_MIXER_Anforderung,
           SpIBit                   := I    270.3);

// A12_FUELLER_CIP_BEREIT SpI 007 Koppelsignal von Füller 12 CIP-Bereitschaft (Dauersignal)
      CALL FC    14 (
           UnitNo                   := #UnitNo,
           SpIRec                   := DB2721.A12_FUELLER_CIP_BEREIT,
           SpIBit                   := I    268.0);

// GOA_1203 SpI 009
      CALL FC    14 (
           UnitNo                   := #UnitNo,
           SpIRec                   := DB2721.GOA_1203,
           SpIBit                   := I    262.2);

// TS_HL_A12 SpI 010
      CALL FC    14 (
           UnitNo                   := #UnitNo,
           SpIRec                   := DB2721.TS_HL_A12,
           SpIBit                   := I     14.4);

// A12_FUELLER_LEER SpI 011 Koppelsignal von Füller 12 Füller leer (Impuls)
      CALL FC    14 (
           UnitNo                   := #UnitNo,
           SpIRec                   := DB2721.A12_FUELLER_LEER,
           SpIBit                   := I    268.2);

// A12_FUELLER_VOLL SpI 012 Koppelsignal von Füller 12 Füller voll (Impuls)
      CALL FC    14 (
           UnitNo                   := #UnitNo,
           SpIRec                   := DB2721.A12_FUELLER_VOLL,
           SpIBit                   := I    268.3);

NETWORK
TITLE =messages

      NOP   0;
// msg001 Msg 001 Message 01
      CALL FC    16 (
           UnitNo                   := #UnitNo,
           MsgRec                   := DB2727.msg001,
           MsgBit                   := DB2727.DBX   82.7);

// msg002 Msg 002 Message 02
      CALL FC    16 (
           UnitNo                   := #UnitNo,
           MsgRec                   := DB2727.msg002,
           MsgBit                   := DB2727.DBX  142.7);

// msg003 Msg 003 Message 03
      CALL FC    16 (
           UnitNo                   := #UnitNo,
           MsgRec                   := DB2727.msg003,
           MsgBit                   := DB2727.DBX  202.7);

NETWORK
TITLE =unit supply

      UC    FB [#UnitFB];

NETWORK
TITLE =A12_RRP1  Reinigungsrücklaufpumpe A12
// Act 001
// Box           : LT-CIP
// Input address : I256.4
// Output address: Q256.4
      CALL FC    70 (
           UnitNo                   := #UnitNo,
           ActRec                   := DB2720.A12_RRP1,
           Typ                      := 1,
           FBa                      := #xTmp,
           FBa2                     := I    256.4,
           Out                      := Q    256.4);

NETWORK
TITLE =F12_Maschine_Start  Füller A12 Maschine Start
// Act 002
// Box           : Füller12
// Output address: Q268.0
      CALL FC    70 (
           UnitNo                   := #UnitNo,
           ActRec                   := DB2720.F12_Maschine_Start,
           Typ                      := 0,
           FBa                      := #xTmp,
           FBa2                     := #xTmp,
           Out                      := Q    268.0);

NETWORK
TITLE =F12_Maschine_Stop  Füller A12 Maschine Stop
// Act 003
// Box           : Füller12
// Output address: Q268.1
      CALL FC    70 (
           UnitNo                   := #UnitNo,
           ActRec                   := DB2720.F12_Maschine_Stop,
           Typ                      := 0,
           FBa                      := #xTmp,
           FBa2                     := #xTmp,
           Out                      := #xTmp);

NETWORK
TITLE =F12_Kreislauf_o_puls  Füller A12 CIP-Kreislauf ohne pulsierenden
// Act 010
// Box           : Füller12
// Output address: Q268.2
      CALL FC    70 (
           UnitNo                   := #UnitNo,
           ActRec                   := DB2720.F12_Kreislauf_o_puls,
           Typ                      := 0,
           FBa                      := #xTmp,
           FBa2                     := #xTmp,
           Out                      := Q    268.2);

NETWORK
TITLE =F12_Kreislauf_m_puls  Füller A12 CIP-Kreislauf mit pulsierenden
// Act 011
// Box           : Füller12
// Output address: Q268.3
      CALL FC    70 (
           UnitNo                   := #UnitNo,
           ActRec                   := DB2720.F12_Kreislauf_m_puls,
           Typ                      := 0,
           FBa                      := #xTmp,
           FBa2                     := #xTmp,
           Out                      := Q    268.3);

NETWORK
TITLE =F12_Randvollstellung  Füller A12 Randvollstellung Standdesinfekt
// Act 012
// Box           : Füller12
// Output address: Q268.4
      CALL FC    70 (
           UnitNo                   := #UnitNo,
           ActRec                   := DB2720.F12_Randvollstellung,
           Typ                      := 0,
           FBa                      := #xTmp,
           FBa2                     := #xTmp,
           Out                      := Q    268.4);

NETWORK
TITLE =F12_Klarspuelen_o_CIP_Be  Füller A12 Klarspülen ohne CIP-Behälte
// Act 013
// Box           : Füller12
// Output address: Q268.5
      CALL FC    70 (
           UnitNo                   := #UnitNo,
           ActRec                   := DB2720.F12_Klarspuelen_o_CIP_Be,
           Typ                      := 0,
           FBa                      := #xTmp,
           FBa2                     := #xTmp,
           Out                      := Q    268.5);

NETWORK
TITLE =F12_Ausschub_m_Sterilluf  Füller A12 Ausschubprogramm mit Steril
// Act 014
// Box           : Füller12
// Output address: Q268.6
      CALL FC    70 (
           UnitNo                   := #UnitNo,
           ActRec                   := DB2720.F12_Ausschub_m_Sterilluf,
           Typ                      := 0,
           FBa                      := #xTmp,
           FBa2                     := #xTmp,
           Out                      := Q    268.6);

NETWORK
TITLE =F12_Ausschub_m_CO2  Füller A12 Ausschubprogramm mit CO2
// Act 015
// Box           : Füller12
// Output address: Q268.7
      CALL FC    70 (
           UnitNo                   := #UnitNo,
           ActRec                   := DB2720.F12_Ausschub_m_CO2,
           Typ                      := 0,
           FBa                      := #xTmp,
           FBa2                     := #xTmp,
           Out                      := Q    268.7);

NETWORK
TITLE =F12_Grundstellung  Füller A12 Maschine Grundstellung (Impuls)
// Act 016
// Box           : Füller12
// Output address: Q269.0
      CALL FC    70 (
           UnitNo                   := #UnitNo,
           ActRec                   := DB2720.F12_Grundstellung,
           Typ                      := 0,
           FBa                      := #xTmp,
           FBa2                     := #xTmp,
           Out                      := Q    269.0);

NETWORK
TITLE =F12_Drainagestellung  Füller A12 Drainagestellung (Impuls)
// Act 017
// Box           : Füller12
// Output address: Q269.1
      CALL FC    70 (
           UnitNo                   := #UnitNo,
           ActRec                   := DB2720.F12_Drainagestellung,
           Typ                      := 0,
           FBa                      := #xTmp,
           FBa2                     := #xTmp,
           Out                      := Q    269.1);

NETWORK
TITLE =F12_Bypass  Füller A12 Bypass (Impuls)
// Act 018
// Box           : Füller12
// Output address: Q269.2
      CALL FC    70 (
           UnitNo                   := #UnitNo,
           ActRec                   := DB2720.F12_Bypass,
           Typ                      := 0,
           FBa                      := #xTmp,
           FBa2                     := #xTmp,
           Out                      := Q    269.2);

NETWORK
TITLE =A12RR1  A12RR1 CIP Rücklaufventil Kreis 1 Anlage 12
// Act 020
// Box           : VS-RRA
// Input address : I200.3
// Output address: Q200.3
      CALL FC    70 (
           UnitNo                   := #UnitNo,
           ActRec                   := DB2720.A12RR1,
           Typ                      := 1,
           FBa                      := #xTmp,
           FBa2                     := I    200.3,
           Out                      := Q    200.3);

NETWORK
TITLE =A12RR2  A12RR1 CIP Rücklaufventil Kreis 2 Anlage 12
// Act 021
// Box           : VS-RRA
// Input address : I200.4
// Output address: Q200.4
      CALL FC    70 (
           UnitNo                   := #UnitNo,
           ActRec                   := DB2720.A12RR2,
           Typ                      := 1,
           FBa                      := #xTmp,
           FBa2                     := I    200.4,
           Out                      := Q    200.4);

NETWORK
TITLE =A12RR3  A12RR1 CIP Rücklaufventil Kreis 3 Anlage 12
// Act 022
// Box           : VS-RRA
// Input address : I200.5
// Output address: Q200.5
      CALL FC    70 (
           UnitNo                   := #UnitNo,
           ActRec                   := DB2720.A12RR3,
           Typ                      := 1,
           FBa                      := #xTmp,
           FBa2                     := I    200.5,
           Out                      := Q    200.5);

NETWORK
TITLE =M12_Grundstellung  Mixer A12 Grundstellung (Impuls)
// Act 023
// Box           : Mixer12
// Output address: Q270.0
      CALL FC    70 (
           UnitNo                   := #UnitNo,
           ActRec                   := DB2720.M12_Grundstellung,
           Typ                      := 0,
           FBa                      := #xTmp,
           FBa2                     := #xTmp,
           Out                      := Q    270.0);

NETWORK
TITLE =M12_Drainagestellung  Mixer A12 Drainagestellung (Impuls)
// Act 024
// Box           : Mixer12
// Output address: Q270.1
      CALL FC    70 (
           UnitNo                   := #UnitNo,
           ActRec                   := DB2720.M12_Drainagestellung,
           Typ                      := 0,
           FBa                      := #xTmp,
           FBa2                     := #xTmp,
           Out                      := Q    270.1);

NETWORK
TITLE =M12_Ausspritzen_o_Ablauf  Mixer A12 Ausspritzen ohne Ablauf (Imp
// Act 025
// Box           : Mixer12
// Output address: Q270.2
      CALL FC    70 (
           UnitNo                   := #UnitNo,
           ActRec                   := DB2720.M12_Ausspritzen_o_Ablauf,
           Typ                      := 0,
           FBa                      := #xTmp,
           FBa2                     := #xTmp,
           Out                      := Q    270.2);

NETWORK
TITLE =M12_Ausspritzen_m_Ablauf  Mixer A12 Ausspritzen mit Ablauf (Impu
// Act 026
// Box           : Mixer12
// Output address: Q270.3
      CALL FC    70 (
           UnitNo                   := #UnitNo,
           ActRec                   := DB2720.M12_Ausspritzen_m_Ablauf,
           Typ                      := 0,
           FBa                      := #xTmp,
           FBa2                     := #xTmp,
           Out                      := Q    270.3);

NETWORK
TITLE =M12_Fluten_o_Ablauf  Mixer A12 Fluten ohne Ablauf (Impuls)
// Act 027
// Box           : Mixer12
// Output address: Q270.4
      CALL FC    70 (
           UnitNo                   := #UnitNo,
           ActRec                   := DB2720.M12_Fluten_o_Ablauf,
           Typ                      := 0,
           FBa                      := #xTmp,
           FBa2                     := #xTmp,
           Out                      := Q    270.4);

NETWORK
TITLE =M12_Fluten_m_Ablauf  Mixer A12 Fluten mit Ablauf (Impuls)
// Act 028
// Box           : Mixer12
// Output address: Q270.5
      CALL FC    70 (
           UnitNo                   := #UnitNo,
           ActRec                   := DB2720.M12_Fluten_m_Ablauf,
           Typ                      := 0,
           FBa                      := #xTmp,
           FBa2                     := #xTmp,
           Out                      := Q    270.5);

NETWORK
TITLE =M12_Randvollstellung  Mixer A12 Randvollstellung (Impuls)
// Act 029
// Box           : Mixer12
// Output address: Q270.6
      CALL FC    70 (
           UnitNo                   := #UnitNo,
           ActRec                   := DB2720.M12_Randvollstellung,
           Typ                      := 0,
           FBa                      := #xTmp,
           FBa2                     := #xTmp,
           Out                      := Q    270.6);

NETWORK
TITLE =M12_Abpumpen  Mixer A12 Abpumpen (Impuls)
// Act 030
// Box           : Mixer12
// Output address: Q270.7
      CALL FC    70 (
           UnitNo                   := #UnitNo,
           ActRec                   := DB2720.M12_Abpumpen,
           Typ                      := 0,
           FBa                      := #xTmp,
           FBa2                     := #xTmp,
           Out                      := Q    270.7);

NETWORK
TITLE =M12_Klarspuelen  Mixer A12 Klarspülen
// Act 031
// Box           : Mixer12
// Output address: Q271.0
      CALL FC    70 (
           UnitNo                   := #UnitNo,
           ActRec                   := DB2720.M12_Klarspuelen,
           Typ                      := 0,
           FBa                      := #xTmp,
           FBa2                     := #xTmp,
           Out                      := Q    271.0);

END_FUNCTION_BLOCK

FUNCTION_BLOCK FB 1721
TITLE =U072: Packaging Plant 12
FAMILY : BOTEC_F1
NAME : UniE
VERSION : 1.2


VAR_TEMP
  CIP : BOOL ;	//CIP active
  UNIM : BOOL ;	//Unit Not In Maintenance
  GenRel : BOOL ;	//general OK (emergency and maintenance OK)
  EStopOK : BOOL ;	//emergency OK
  UnitNo : INT ;	//unit number
  xTmp : BOOL ;	//Temporary Bool
  iTmp : INT ;	//Temporary INT
  rTmp : REAL ;	//Temporary REAL
  dTmp : DINT ;	//Temporary DINT (free for general use)
  RetValInt : INT ;	//return value
END_VAR
BEGIN
NETWORK
TITLE =General

      SET   ;
// Simulation ---------------------------------------------------------------
      A     DB1721.DBX 1357.7;
      CC    FB  1729; // "U072Sim"
      A     DB1721.DBX   17.3;
      =     DB1721.DBX 1357.7; //Help bit for simulation

// get unit number ----------------------------------------------------------
      L     DB1720.DBW    0;
      T     #UnitNo;

// CIP ----------------------------------------------------------------------
      L     DB1721.DBD   54;
      L     0;
      <D    ;
      =     #CIP;

// emergency OK -------------------------------------------------------------
      A     DB1725.DBX   27.0; //Emergency Stop OK
      =     #EStopOK;

// Write Unit in Maintenance ------------------------------------------------

      AN    DB1721.DBX   69.7;
      =     #UNIM;

// emergency and maintenance OK ---------------------------------------------
      A     #EStopOK;
      A     #UNIM;
      =     #GenRel;

// communication ------------------------------------------------------------
      UC    FB  1725; // U072Com

NETWORK
TITLE =Universal Value

      NOP   0;

// ----------------------------------------------------------
// unv001 Process Status
// ----------------------------------------------------------
// process value to UnV
//      L     0.000000e+000
//      T     "U072UnVD".unv001.ValExt

// ----------------------------------------------------------
// unv002 Universal Value 02
// ----------------------------------------------------------
// process value to UnV
//      L     0.000000e+000
//      T     "U072UnVD".unv002.ValExt

// ----------------------------------------------------------
// unv003 Universal Value 03
// ----------------------------------------------------------
// process value to UnV
//      L     0.000000e+000
//      T     "U072UnVD".unv003.ValExt

// ----------------------------------------------------------
// unv004 Universal Value 04
// ----------------------------------------------------------
// process value to UnV
//      L     0.000000e+000
//      T     "U072UnVD".unv004.ValExt

NETWORK
TITLE =Special Input

      NOP   0;
// ----------------------------------------------------------
// A12_FS1
// ----------------------------------------------------------
      A     DB2720.DBX  102.6;
      =     DB2721.DBX   81.4;
//      =     "U072SpID".A12_FS1.Pre

// ----------------------------------------------------------
// GOA_1203
// ----------------------------------------------------------
//     A     "U072SeqD".Seq.Step0
//      A     #CIP
//      =     "U072SpID".GOA_1203.EAl
//     =     "U072SpID".GOA_1203.Pre

// ----------------------------------------------------------
// TS_HL_A12
// ----------------------------------------------------------
//      CLR
//      =     "U072SpID".TS_HL_A12.EAl
//      =     "U072SpID".TS_HL_A12.Pre

// ----------------------------------------------------------
// A12A_E_CIP_BEREIT SIGNAL VON FUELLER 6A
// ----------------------------------------------------------
//      CLR
//      =     "U072SpID".A12A_E_CIP_BEREIT.EAl
//     =     "U072SpID".A12A_E_CIP_BEREIT.Pre

// ----------------------------------------------------------
// A12A_E_LEER_MEDIENWECHSE SIGNAL VON FUELLER 6A
// ----------------------------------------------------------
//      CLR
//      =     "U072SpID".A12A_E_LEER_MEDIENWECHSE.EAl
//     =     "U072SpID".A12A_E_LEER_MEDIENWECHSE.Pre
//
// ----------------------------------------------------------
// A12A_E_MIX_CIP_BEREIT SIGNAL VON FUELLER 6A
// ----------------------------------------------------------
//      CLR
//      =     "U072SpID".A12A_E_MIX_CIP_BEREIT.EAl
//     =     "U072SpID".A12A_E_MIX_CIP_BEREIT.Pre

// ----------------------------------------------------------
// A12A_E_MIX_HALT SIGNAL VON FUELLER 6A
// ----------------------------------------------------------
//      CLR
//     =     "U072SpID".A12A_E_MIX_HALT.EAl
//     =     "U072SpID".A12A_E_MIX_HALT.Pre

// ----------------------------------------------------------
// A12A_E_WASSERANFORDERUNG SIGNAL VON FUELLER 6A
// ----------------------------------------------------------
//      CLR
//      =     "U072SpID".A12A_E_WASSERANFORDERUNG.EAl
//      =     "U072SpID".A12A_E_WASSERANFORDERUNG.Pre

// ----------------------------------------------------------
// RM_A12RP2 SIGNAL VON FUELLER 6A
// ----------------------------------------------------------
//      CLR
//      =     "U072SpID".RM_A12RP2.EAl
//      =     "U072SpID".RM_A12RP2.Pre

NETWORK
TITLE =Messages

      NOP   0;

// ----------------------------------------------------------
// msg001 Message 01
// ----------------------------------------------------------
      SET   ;
      R     DB2727.DBX   80.7;
      =     DB2727.DBX   81.4;

      CLR   ;
      =     DB2727.DBX   82.7;

// ----------------------------------------------------------
// msg002 Message 02
// ----------------------------------------------------------
      SET   ;
      R     DB2727.DBX  140.7;
      =     DB2727.DBX  141.4;

      CLR   ;
      =     DB2727.DBX  142.7;

// ----------------------------------------------------------
// msg003 Message 03
// ----------------------------------------------------------
      SET   ;
      R     DB2727.DBX  200.7;
      =     DB2727.DBX  201.4;

      CLR   ;
      =     DB2727.DBX  202.7;

NETWORK
TITLE =Sequence organisation

      CLR   ;
      =     M    122.2;

// SFM supply ----------------------------------------------------------------

// sequencer ----------------------------------------------------------------
      A     DB1723.DBX   43.1;
      S     DB1723.DBX   97.3;

      CALL FC    40 (
           UnitNo                   := #UnitNo);

NETWORK
TITLE =Auto / Manual

      SET   ;
      AN    M    122.2;
      JC    MODE;
      AN    M    120.1;

// assign actuator mode
      AN    M    120.1;
      =     DB2720.DBX  105.4;
      =     DB2720.DBX  185.4;
      S     DB2720.DBX  265.4;
      =     DB2720.DBX  345.4;
      =     DB2720.DBX  425.4;
      =     DB2720.DBX  505.4;
      =     DB2720.DBX  585.4;
      =     DB2720.DBX  665.4;
      =     DB2720.DBX  745.4;
      =     DB2720.DBX  825.4;
      =     DB2720.DBX  905.4;
      =     DB2720.DBX  985.4;
      =     DB2720.DBX 1065.4;
      =     DB2720.DBX 1145.4;
      =     DB2720.DBX 1225.4;
      =     DB2720.DBX 1305.4;
      =     DB2720.DBX 1385.4;
      =     DB2720.DBX 1465.4;

      =     DB2720.DBX 1625.4;
      =     DB2720.DBX 1705.4;
      =     DB2720.DBX 1785.4;

      =     DB2720.DBX 1865.4;
      =     DB2720.DBX 1945.4;
      =     DB2720.DBX 2025.4;
      =     DB2720.DBX 2105.4;
      =     DB2720.DBX 2185.4;
      =     DB2720.DBX 2265.4;
      =     DB2720.DBX 2345.4;
      =     DB2720.DBX 2425.4;
      =     DB2720.DBX 2505.4;


MODE: SET   ;

NETWORK
TITLE =RWPA12 Pumpe --> Anlage 12
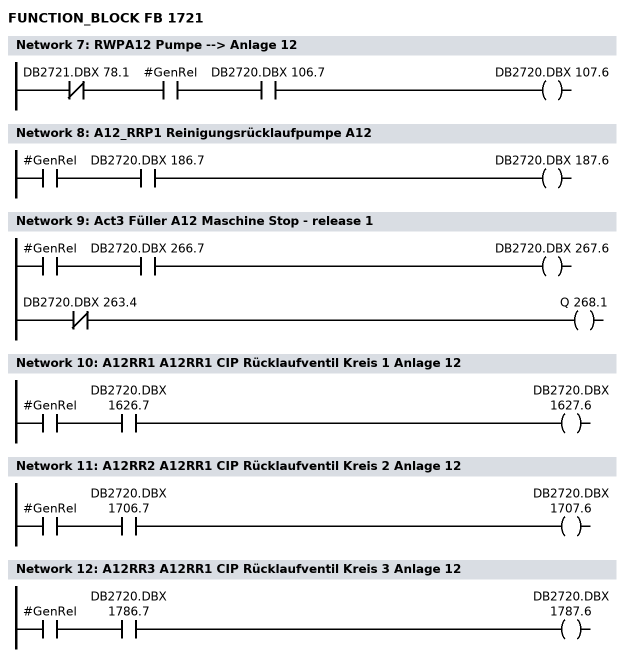

      AN    DB2721.DBX   78.1;

      A     #GenRel;
      A     DB2720.DBX  106.7;
      =     DB2720.DBX  107.6;
NETWORK
TITLE =A12_RRP1 Reinigungsrücklaufpumpe A12

      A     #GenRel;
      A     DB2720.DBX  186.7;
      =     DB2720.DBX  187.6;

NETWORK
TITLE =Act3 Füller A12 Maschine Stop - release 1

      A     #GenRel;
      A     DB2720.DBX  266.7;
      =     DB2720.DBX  267.6;

      AN    DB2720.DBX  263.4;
      =     Q    268.1;

NETWORK
TITLE =A12RR1 A12RR1 CIP Rücklaufventil Kreis 1 Anlage 12

      A     #GenRel;
      A     DB2720.DBX 1626.7;
      =     DB2720.DBX 1627.6;
NETWORK
TITLE =A12RR2 A12RR1 CIP Rücklaufventil Kreis 2 Anlage 12

      A     #GenRel;
      A     DB2720.DBX 1706.7;
      =     DB2720.DBX 1707.6;
NETWORK
TITLE =A12RR3 A12RR1 CIP Rücklaufventil Kreis 3 Anlage 12

      A     #GenRel;
      A     DB2720.DBX 1786.7;
      =     DB2720.DBX 1787.6;
END_FUNCTION_BLOCK

FUNCTION_BLOCK FB 1740
TITLE =U074: Abfüllanlage 14
FAMILY : BOTEC_F1
NAME : U074A
VERSION : 2.1


VAR_TEMP
  EStopOK : BOOL ;	//auxiliary flag
  CIP : BOOL ;	//CIP Program Selected
  xTmp : BOOL ;	//Temporary Bool(free for general use)
  DummyBool : BOOL ;	//Temporary Bool(free for general use)
  UnitNo : INT ;	//unit number
  UnitFB : INT ;	//unit expansion FB number
  rTmp : REAL ;	//Temporary REAL (free for general use)
  iTmp : INT ;	//Temporary INT (free for general use)
  DummyInt : INT ;	//Temporary INT (free for general use)
  dTmp : DINT ;	//Temporary DINT (free for general use)
END_VAR
BEGIN
NETWORK
TITLE =general

      CLR   ;
      =     #xTmp;
      =     #EStopOK;

      L     DB1740.DBW    0;
      T     #UnitNo;
      L     DB1740.DBW    2;
      T     #UnitFB;

NETWORK
TITLE =analog inputs

      NOP   0;
// U74_AnI001 AnI 001 spare
      CALL FC    24 (
           UnitNo                   := #UnitNo,
           AnIRec                   := DB2743.U74_AnI001,
           ValPer                   := #DummyInt);

// U74_AnI002 AnI 002 spare
      CALL FC    24 (
           UnitNo                   := #UnitNo,
           AnIRec                   := DB2743.U74_AnI002,
           ValPer                   := #DummyInt);

// U74_AnI003 AnI 003 spare
      CALL FC    24 (
           UnitNo                   := #UnitNo,
           AnIRec                   := DB2743.U74_AnI003,
           ValPer                   := #DummyInt);

// U74_AnI004 AnI 004 spare
      CALL FC    24 (
           UnitNo                   := #UnitNo,
           AnIRec                   := DB2743.U74_AnI004,
           ValPer                   := #DummyInt);

// U74_AnI005 AnI 005 spare
      CALL FC    24 (
           UnitNo                   := #UnitNo,
           AnIRec                   := DB2743.U74_AnI005,
           ValPer                   := #DummyInt);

// U74_AnI006 AnI 006 spare
      CALL FC    24 (
           UnitNo                   := #UnitNo,
           AnIRec                   := DB2743.U74_AnI006,
           ValPer                   := #DummyInt);

NETWORK
TITLE =Universal value

      NOP   0;
// unv001 UnV 001 Process Status
      CALL FC    27 (
           UnitNo                   := #UnitNo,
           UnVRec                   := DB2745.unv001,
           ValExt                   := DB2745.DBD  234);

// A14M_PROGRAMM_NR UnV 002 Select programme as number 101 ... 131 instead of bits
      CALL FC    27 (
           UnitNo                   := #UnitNo,
           UnVRec                   := DB2745.A14M_PROGRAMM_NR,
           ValExt                   := DB2745.DBD  362);

// A14M_TANKNR UnV 003 Actual Water Tank
      CALL FC    27 (
           UnitNo                   := #UnitNo,
           UnVRec                   := DB2745.A14M_TANKNR,
           ValExt                   := DB2745.DBD  490);

// A14M_TANKNIVEAU UnV 004 Water Tank Level
      CALL FC    27 (
           UnitNo                   := #UnitNo,
           UnVRec                   := DB2745.A14M_TANKNIVEAU,
           ValExt                   := DB2745.DBD  618);

NETWORK
TITLE =special inputs

      NOP   0;
// A14FS1 SpI 001 Flow Switch RL Anlage 14
      CALL FC    14 (
           UnitNo                   := #UnitNo,
           SpIRec                   := DB2741.A14FS1,
           SpIBit                   := I     99.0);

// A14FR_LAEUFT SpI 002
      CALL FC    14 (
           UnitNo                   := #UnitNo,
           SpIRec                   := DB2741.A14FR_LAEUFT,
           SpIBit                   := I    922.2);

// A14M_CIP_BEREIT SpI 003 Mixer ist Bereit zur Ansteuerung durch die CIP Anlage und hat keine Störung
      CALL FC    14 (
           UnitNo                   := #UnitNo,
           SpIRec                   := DB2741.A14M_CIP_BEREIT,
           SpIBit                   := I    910.1);

// A14M_MIXER_VOLL SpI 004 Alle Tanks und Leitungen sind gefüllt
      CALL FC    14 (
           UnitNo                   := #UnitNo,
           SpIRec                   := DB2741.A14M_MIXER_VOLL,
           SpIBit                   := I    910.3);

// A14M_MIXER_LEER SpI 005 Mixer ist komplett leer
      CALL FC    14 (
           UnitNo                   := #UnitNo,
           SpIRec                   := DB2741.A14M_MIXER_LEER,
           SpIBit                   := I    910.2);

// A14M_ANFORDERUNG_SIRUP SpI 006
      CALL FC    14 (
           UnitNo                   := #UnitNo,
           SpIRec                   := DB2741.A14M_ANFORDERUNG_SIRUP,
           SpIBit                   := I    912.3);

// A14FR_CIP_BEREIT SpI 007
      CALL FC    14 (
           UnitNo                   := #UnitNo,
           SpIRec                   := DB2741.A14FR_CIP_BEREIT,
           SpIBit                   := I    922.1);

// A14FR_WATCHDOG SpI 009
      CALL FC    14 (
           UnitNo                   := #UnitNo,
           SpIRec                   := DB2741.A14FR_WATCHDOG,
           SpIBit                   := I    923.7);

// A14M_WATCHDOG SpI 010
      CALL FC    14 (
           UnitNo                   := #UnitNo,
           SpIRec                   := DB2741.A14M_WATCHDOG,
           SpIBit                   := I    911.7);

// A14FR_LEER SpI 011
      CALL FC    14 (
           UnitNo                   := #UnitNo,
           SpIRec                   := DB2741.A14FR_LEER,
           SpIBit                   := I    922.3);

// A14FR_VOLL SpI 012
      CALL FC    14 (
           UnitNo                   := #UnitNo,
           SpIRec                   := DB2741.A14FR_VOLL,
           SpIBit                   := I    922.4);

// A14FR_DIAGNOSE SpI 015 DP Koppler
      CALL FC    14 (
           UnitNo                   := #UnitNo,
           SpIRec                   := DB2741.A14FR_DIAGNOSE,
           SpIBit                   := I    922.0);

// A14M_STOERUNG_MIXER SpI 016 Störung Mixer
      CALL FC    14 (
           UnitNo                   := #UnitNo,
           SpIRec                   := DB2741.A14M_STOERUNG_MIXER,
           SpIBit                   := I    911.3);

// GOA_1403 SpI 025
      CALL FC    14 (
           UnitNo                   := #UnitNo,
           SpIRec                   := DB2741.GOA_1403,
           SpIBit                   := I     98.2);

NETWORK
TITLE =messages

      NOP   0;
// msg001 Msg 001 Message 01
      CALL FC    16 (
           UnitNo                   := #UnitNo,
           MsgRec                   := DB2747.msg001,
           MsgBit                   := DB2747.DBX   82.7);

// msg002 Msg 002 Message 02
      CALL FC    16 (
           UnitNo                   := #UnitNo,
           MsgRec                   := DB2747.msg002,
           MsgBit                   := DB2747.DBX  142.7);

// msg003 Msg 003 Message 03
      CALL FC    16 (
           UnitNo                   := #UnitNo,
           MsgRec                   := DB2747.msg003,
           MsgBit                   := DB2747.DBX  202.7);

NETWORK
TITLE =unit supply

      UC    FB [#UnitFB];

NETWORK
TITLE =A14RRP1  Reinigungsrücklaufpumpe Anlage 14
// Act 001
// Box           : VSA14
// Input address : I97.7
// Output address: Q97.7
      CALL FC    70 (
           UnitNo                   := #UnitNo,
           ActRec                   := DB2740.A14RRP1,
           Typ                      := 1,
           FBa                      := #xTmp,
           FBa2                     := I     97.7,
           Out                      := Q     97.7);

NETWORK
TITLE =A14FR_START
// Act 002
// Box           : A14 Füller|Rinser
// Output address: Q922.1
      CALL FC    70 (
           UnitNo                   := #UnitNo,
           ActRec                   := DB2740.A14FR_START,
           Typ                      := 0,
           FBa                      := #xTmp,
           FBa2                     := #xTmp,
           Out                      := Q    922.1);

NETWORK
TITLE =A14FR_STOP
// Act 003
// Box           : A14 Füller|Rinser
// Output address: Q922.2
      CALL FC    70 (
           UnitNo                   := #UnitNo,
           ActRec                   := DB2740.A14FR_STOP,
           Typ                      := 0,
           FBa                      := #xTmp,
           FBa2                     := #xTmp,
           Out                      := #xTmp);

NETWORK
TITLE =A14FR_KREISLAUF_OHNE_ABL  CIP Kreislauf ohne pulsierendem Ablauf
// Act 010
// Box           : A14 Füller|Rinser
// Output address: Q922.5
      CALL FC    70 (
           UnitNo                   := #UnitNo,
           ActRec                   := DB2740.A14FR_KREISLAUF_OHNE_ABL,
           Typ                      := 0,
           FBa                      := #xTmp,
           FBa2                     := #xTmp,
           Out                      := Q    922.5);

NETWORK
TITLE =A14FR_KREISLAUF_MIT_ABLA  CIP Kreislauf mit pulsierendem Ablauf
// Act 011
// Box           : A14 Füller|Rinser
// Output address: Q922.6
      CALL FC    70 (
           UnitNo                   := #UnitNo,
           ActRec                   := DB2740.A14FR_KREISLAUF_MIT_ABLA,
           Typ                      := 0,
           FBa                      := #xTmp,
           FBa2                     := #xTmp,
           Out                      := Q    922.6);

NETWORK
TITLE =A14FR_RANDVOLLSTELLUNG  Randvollstellung
// Act 012
// Box           : A14 Füller|Rinser
// Output address: Q923.1
      CALL FC    70 (
           UnitNo                   := #UnitNo,
           ActRec                   := DB2740.A14FR_RANDVOLLSTELLUNG,
           Typ                      := 0,
           FBa                      := #xTmp,
           FBa2                     := #xTmp,
           Out                      := Q    923.1);

NETWORK
TITLE =A14FR_KLARSPUELEN  Klarspülen
// Act 013
// Box           : A14 Füller|Rinser
// Output address: Q923.2
      CALL FC    70 (
           UnitNo                   := #UnitNo,
           ActRec                   := DB2740.A14FR_KLARSPUELEN,
           Typ                      := 0,
           FBa                      := #xTmp,
           FBa2                     := #xTmp,
           Out                      := Q    923.2);

NETWORK
TITLE =A14FR_AUSSCHUB_M_STERILL  Ausschub mit Sterilluft
// Act 014
// Box           : A14 Füller|Rinser
// Output address: Q922.7
      CALL FC    70 (
           UnitNo                   := #UnitNo,
           ActRec                   := DB2740.A14FR_AUSSCHUB_M_STERILL,
           Typ                      := 0,
           FBa                      := #xTmp,
           FBa2                     := #xTmp,
           Out                      := Q    922.7);

NETWORK
TITLE =A14FR_AUSSCHUB_M_CO2  Ausschub mit CO2
// Act 015
// Box           : A14 Füller|Rinser
// Output address: Q923.3
      CALL FC    70 (
           UnitNo                   := #UnitNo,
           ActRec                   := DB2740.A14FR_AUSSCHUB_M_CO2,
           Typ                      := 0,
           FBa                      := #xTmp,
           FBa2                     := #xTmp,
           Out                      := Q    923.3);

NETWORK
TITLE =A14FR_GRUNDSTELLUNG  Grundstellung
// Act 016
// Box           : A14 Füller|Rinser
// Output address: Q922.3
      CALL FC    70 (
           UnitNo                   := #UnitNo,
           ActRec                   := DB2740.A14FR_GRUNDSTELLUNG,
           Typ                      := 0,
           FBa                      := #xTmp,
           FBa2                     := #xTmp,
           Out                      := Q    922.3);

NETWORK
TITLE =A14FR_DRAINAGE  Drainagestellung
// Act 017
// Box           : A14 Füller|Rinser
// Output address: Q922.4
      CALL FC    70 (
           UnitNo                   := #UnitNo,
           ActRec                   := DB2740.A14FR_DRAINAGE,
           Typ                      := 0,
           FBa                      := #xTmp,
           FBa2                     := #xTmp,
           Out                      := Q    922.4);

NETWORK
TITLE =A14FR_BYPASS  Bypass
// Act 018
// Box           : A14 Füller|Rinser
// Output address: Q923.0
      CALL FC    70 (
           UnitNo                   := #UnitNo,
           ActRec                   := DB2740.A14FR_BYPASS,
           Typ                      := 0,
           FBa                      := #xTmp,
           FBa2                     := #xTmp,
           Out                      := Q    923.0);

NETWORK
TITLE =A14_RR1
// Act 020
// Box           : VS-RRA
// Input address : I201.5
// Output address: Q201.5
      CALL FC    70 (
           UnitNo                   := #UnitNo,
           ActRec                   := DB2740.A14_RR1,
           Typ                      := 1,
           FBa                      := #xTmp,
           FBa2                     := I    201.5,
           Out                      := Q    201.5);

NETWORK
TITLE =A14_RR2
// Act 021
// Box           : VS-RRA
// Input address : I201.6
// Output address: Q201.6
      CALL FC    70 (
           UnitNo                   := #UnitNo,
           ActRec                   := DB2740.A14_RR2,
           Typ                      := 1,
           FBa                      := #xTmp,
           FBa2                     := I    201.6,
           Out                      := Q    201.6);

NETWORK
TITLE =A14_RR3
// Act 022
// Box           : VS-RRA
// Input address : I201.7
// Output address: Q201.7
      CALL FC    70 (
           UnitNo                   := #UnitNo,
           ActRec                   := DB2740.A14_RR3,
           Typ                      := 1,
           FBa                      := #xTmp,
           FBa2                     := I    201.7,
           Out                      := Q    201.7);

NETWORK
TITLE =A14M_GRUNDSTELLUNG
// Act 023
// Box           : A14 Mixer
// Output address: Q910.1
      CALL FC    70 (
           UnitNo                   := #UnitNo,
           ActRec                   := DB2740.A14M_GRUNDSTELLUNG,
           Typ                      := 0,
           FBa                      := #xTmp,
           FBa2                     := #xTmp,
           Out                      := Q    910.1);

NETWORK
TITLE =A14M_DRAINAGE  Drainage
// Act 024
// Box           : A14 Mixer
// Output address: Q910.2
      CALL FC    70 (
           UnitNo                   := #UnitNo,
           ActRec                   := DB2740.A14M_DRAINAGE,
           Typ                      := 0,
           FBa                      := #xTmp,
           FBa2                     := #xTmp,
           Out                      := Q    910.2);

NETWORK
TITLE =A14M_AUSSPRITZEN_OHNE_AB  Ausspritzen ohne Ablauf
// Act 025
// Box           : A14 Mixer
// Output address: Q910.4
      CALL FC    70 (
           UnitNo                   := #UnitNo,
           ActRec                   := DB2740.A14M_AUSSPRITZEN_OHNE_AB,
           Typ                      := 0,
           FBa                      := #xTmp,
           FBa2                     := #xTmp,
           Out                      := Q    910.4);

NETWORK
TITLE =A14M_AUSSPRITZEN_MIT_ABL  Ausspritzen mit Ablauf
// Act 026
// Box           : A14 Mixer
// Output address: Q910.5
      CALL FC    70 (
           UnitNo                   := #UnitNo,
           ActRec                   := DB2740.A14M_AUSSPRITZEN_MIT_ABL,
           Typ                      := 0,
           FBa                      := #xTmp,
           FBa2                     := #xTmp,
           Out                      := Q    910.5);

NETWORK
TITLE =A14M_RANDVOLLSTELLUNG  Fluten und Randvollstellung
// Act 029
// Box           : A14 Mixer
// Output address: Q910.7
      CALL FC    70 (
           UnitNo                   := #UnitNo,
           ActRec                   := DB2740.A14M_RANDVOLLSTELLUNG,
           Typ                      := 0,
           FBa                      := #xTmp,
           FBa2                     := #xTmp,
           Out                      := Q    910.7);

NETWORK
TITLE =A14M_ABPUMPEN_MIT_VAKUUM  Abpumpen mit Vakuumausgleich
// Act 030
// Box           : A14 Mixer
// Output address: Q910.6
      CALL FC    70 (
           UnitNo                   := #UnitNo,
           ActRec                   := DB2740.A14M_ABPUMPEN_MIT_VAKUUM,
           Typ                      := 0,
           FBa                      := #xTmp,
           FBa2                     := #xTmp,
           Out                      := Q    910.6);

NETWORK
TITLE =A14M_DRAINAGE_M_VAKUUMAU  Drainage mit Vakuumausgleich
// Act 032
// Box           : A14 Mixer
// Output address: Q910.3
      CALL FC    70 (
           UnitNo                   := #UnitNo,
           ActRec                   := DB2740.A14M_DRAINAGE_M_VAKUUMAU,
           Typ                      := 0,
           FBa                      := #xTmp,
           FBa2                     := #xTmp,
           Out                      := Q    910.3);

NETWORK
TITLE =A14M_STERILISATION
// Act 033
// Box           : A14 Mixer
// Output address: Q911.0
      CALL FC    70 (
           UnitNo                   := #UnitNo,
           ActRec                   := DB2740.A14M_STERILISATION,
           Typ                      := 0,
           FBa                      := #xTmp,
           FBa2                     := #xTmp,
           Out                      := Q    911.0);

END_FUNCTION_BLOCK

FUNCTION_BLOCK FB 1741
TITLE =U074: Packaging Plant 14
FAMILY : BOTEC_F1
NAME : UniE
VERSION : 1.2


VAR_TEMP
  CIP : BOOL ;	//CIP active
  UNIM : BOOL ;	//Unit Not In Maintenance
  GenRel : BOOL ;	//general OK (emergency and maintenance OK)
  EStopOK : BOOL ;	//emergency OK
  UnitNo : INT ;	//unit number
  xTmp : BOOL ;	//Temporary Bool
  iTmp : INT ;	//Temporary INT
  rTmp : REAL ;	//Temporary REAL
  dTmp : DINT ;	//Temporary DINT (free for general use)
  RetValInt : INT ;	//return value
END_VAR
BEGIN
NETWORK
TITLE =General

      SET   ;
// Simulation ---------------------------------------------------------------
      A     DB1741.DBX 1357.7;
      CC    FB  1749; // "U074Sim"
      A     DB1741.DBX   17.3;
      =     DB1741.DBX 1357.7; //Help bit for simulation

// get unit number ----------------------------------------------------------
      L     DB1740.DBW    0;
      T     #UnitNo;

// CIP ----------------------------------------------------------------------
      L     DB1741.DBD   54;
      L     0;
      <D    ;
      =     #CIP;

// emergency OK -------------------------------------------------------------
      A     DB1745.DBX   27.0; //Emergency Stop OK
      =     #EStopOK;

// Write Unit in Maintenance ------------------------------------------------

      AN    DB1741.DBX   69.7;
      =     #UNIM;

// emergency and maintenance OK ---------------------------------------------
      A     #EStopOK;
      A     #UNIM;
      =     #GenRel;

// communication ------------------------------------------------------------
      UC    FB  1745; // U074Com

NETWORK
TITLE =Analog Inputs

      NOP   0;

// ----------------------------------------------------------
// U74_AnI001 spare
// ----------------------------------------------------------
      L     IW   914;
      ITD   ;
      DTR   ;
      T     DB2743.DBD  214;
      SET   ;
      =     DB2743.DBX  143.5;

      L     DB1741.DBD 1118; // !!! insert correct SFM !!!
      T     DB2743.DBD  238;

      SET   ;
      =     DB2743.DBX  141.5;

NETWORK
TITLE =Universal Value

      NOP   0;

// ----------------------------------------------------------
// unv001 Process Status
// ----------------------------------------------------------
// process value to UnV
//      L     0.000000e+000
//      T     "U074UnVD".unv001.ValExt

// ----------------------------------------------------------
// A14M_PROGRAMM_NR Select programme as number 101 ... 131 instead of bits
// ----------------------------------------------------------
// process value to UnV
//      L     0.000000e+000
//      T     "U074UnVD".A14M_PROGRAMM_NR.ValExt

// ----------------------------------------------------------
// A14M_TANKNR Actual Water Tank
// ----------------------------------------------------------
// process value to UnV
//      L     0.000000e+000
//      T     "U074UnVD".A14M_TANKNR.ValExt

// ----------------------------------------------------------
// A14M_TANKNIVEAU Water Tank Level
// ----------------------------------------------------------
// process value to UnV
//      L     0.000000e+000
//      T     "U074UnVD".A14M_TANKNIVEAU.ValExt

NETWORK
TITLE =Special Input

      NOP   0;

// ----------------------------------------------------------
// A14FS1 Flow Switch RL Anlage 14
// ----------------------------------------------------------
//      CLR
//      =     "U074SpID".A14FS1.EAl
//      =     "U074SpID".A14FS1.Pre

// ----------------------------------------------------------
// GOA_1403
// ----------------------------------------------------------
//      CLR
//      =     "U074SpID".A14FR_LAEUFT.EAl
//      =     "U074SpID".A14FR_LAEUFT.Pre

// ----------------------------------------------------------
// A14_FREIGABE_MOLCH_SS
// ----------------------------------------------------------
//      CLR
//      =     "U074SpID".A14_FREIGABE_MOLCH_SS.EAl
//      =     "U074SpID".A14_FREIGABE_MOLCH_SS.Pre

// ----------------------------------------------------------
// A14_MOLCH_STOP_DT
// ----------------------------------------------------------
//      CLR
//      =     "U074SpID".A14_MOLCH_STOP_DT.EAl
//      =     "U074SpID".A14_MOLCH_STOP_DT.Pre


NETWORK
TITLE =Messages

      NOP   0;

// ----------------------------------------------------------
// msg001 Message 01
// ----------------------------------------------------------
      SET   ;
      R     DB2747.DBX   80.7;
      =     DB2747.DBX   81.4;

      CLR   ;
      =     DB2747.DBX   82.7;

// ----------------------------------------------------------
// msg002 Message 02
// ----------------------------------------------------------
      SET   ;
      R     DB2747.DBX  140.7;
      =     DB2747.DBX  141.4;

      CLR   ;
      =     DB2747.DBX  142.7;

// ----------------------------------------------------------
// msg003 Message 03
// ----------------------------------------------------------
      SET   ;
      R     DB2747.DBX  200.7;
      =     DB2747.DBX  201.4;

      CLR   ;
      =     DB2747.DBX  202.7;

NETWORK
TITLE =Sequence organisation

      CLR   ;
      =     M    122.2;

// SFM supply ----------------------------------------------------------------

// analog value to SFM spare -----------------------
      L     DB2743.DBD  146;
      T     DB1741.DBD 1122; // !!! insert correct SFM !!!

// analog value to SFM spare -----------------------
      L     DB2743.DBD  266;
      T     DB1741.DBD 1122; // !!! insert correct SFM !!!

// analog value to SFM spare -----------------------
      L     DB2743.DBD  386;
      T     DB1741.DBD 1122; // !!! insert correct SFM !!!

// analog value to SFM spare -----------------------
      L     DB2743.DBD  506;
      T     DB1741.DBD 1122; // !!! insert correct SFM !!!

// analog value to SFM spare -----------------------
      L     DB2743.DBD  626;
      T     DB1741.DBD 1122; // !!! insert correct SFM !!!

// analog value to SFM spare -----------------------
      L     DB2743.DBD  746;
      T     DB1741.DBD 1122; // !!! insert correct SFM !!!

// sequencer ----------------------------------------------------------------
      A     DB1743.DBX   43.1;
      S     DB1743.DBX   97.3;

      CALL FC    40 (
           UnitNo                   := #UnitNo);

NETWORK
TITLE =Auto / Manual

      SET   ;
      AN    M    122.2;
      JC    MODE;
      AN    M    120.1;

